SPLINE
SPL {X  -124.054, Y  +777.532, Z    +0.000, E1   -54.436, E3 +80490.887}
SPL {X  -145.922, Y  +742.101, Z    +0.000, E1   -46.535, E3 +80509.157}
SPL {X  -155.216, Y  +715.293, Z    +0.000, E1   -34.460, E3 +80515.349}
SPL {X  -159.282, Y  +691.530, Z    +0.000, E1   -17.100, E3 +80518.044}
SPL {X  -159.981, Y  +678.202, Z    +0.000, E1    -4.129, E3 +80518.618}
SPL {X  -159.990, Y  +674.500, Z    +0.000, E1    +0.000, E3 +80518.655}
SPL {X  -159.990, Y  +672.677, Z    +0.000, E1    +3.879, E3 +80518.671}
SPL {X  -159.990, Y  +669.117, Z    +0.000, E1   +12.900, E3 +80518.754}
SPL {X  -159.990, Y  +665.253, Z    +0.000, E1   +22.908, E3 +80518.927}
SPL {X  -159.990, Y  +658.335, Z    +0.000, E1   +38.839, E3 +80519.472}
SPL {X  -159.990, Y  +645.786, Z    +0.000, E1   +56.338, E3 +80521.186}
SPL {X  -159.990, Y  +623.264, Z    +0.000, E1   +67.753, E3 +80526.112}
SPL {X  -159.990, Y  +547.268, Z    +0.000, E1   +73.735, E3 +80551.800}
SPL {X  -159.626, Y  +366.721, Z    +0.000, E1   +74.756, E3 +80634.065}
SPL {X  -157.975, Y  +352.185, Z    +0.000, E1   +74.622, E3 +80644.131}
SPL {X  -154.546, Y  +336.120, Z    +0.000, E1   +74.400, E3 +80655.790}
SPL {X  -141.909, Y  +303.617, Z    +0.000, E1   +76.515, E3 +80650.757}
ENDSPLINE

SPLINE
SPL {X  -142.567, Y  +304.895, Z    +0.000, E1   +75.566, E3 +80659.572}
ENDSPLINE

SPLINE
SPL {X  -141.999, Y  +303.790, Z    +0.000, E1   +74.633, E3 +80668.823}
SPL {X  -141.780, Y  +303.371, Z    +0.000, E1   +73.549, E3 +80678.397}
SPL {X  -140.619, Y  +301.190, Z    +0.000, E1   +72.741, E3 +80686.243}
SPL {X  -137.438, Y  +295.601, Z    +0.000, E1   +72.365, E3 +80692.332}
SPL {X  -134.156, Y  +290.328, Z    +0.000, E1   +71.962, E3 +80698.203}
SPL {X  -130.677, Y  +285.194, Z    +0.000, E1   +71.519, E3 +80704.008}
SPL {X  -127.147, Y  +280.390, Z    +0.000, E1   +71.042, E3 +80709.492}
SPL {X  -123.431, Y  +275.709, Z    +0.000, E1   +70.518, E3 +80714.815}
SPL {X  -120.392, Y  +272.131, Z    +0.000, E1   +70.053, E3 +80718.835}
SPL {X   -79.311, Y  +238.552, Z    +0.000, E1   +58.563, E3 +80814.074}
ENDSPLINE

SPLINE
SPL {X  -105.077, Y  +256.854, Z    +0.000, E1   +55.187, E3 +81001.627}
SPL {X  -133.208, Y  +288.886, Z    +0.000, E1   +52.003, E3 +81034.728}
SPL {X  -149.825, Y  +321.381, Z    +0.000, E1   +42.580, E3 +81047.881}
SPL {X  -156.491, Y  +344.222, Z    +0.000, E1   +30.612, E3 +81052.387}
SPL {X  -159.275, Y  +362.387, Z    +0.000, E1   +16.907, E3 +81054.301}
SPL {X  -159.964, Y  +374.630, Z    +0.000, E1    +5.249, E3 +81054.875}
SPL {X  -159.990, Y  +379.735, Z    +0.000, E1    -0.236, E3 +81054.932}
SPL {X  -159.990, Y  +384.648, Z    +0.000, E1   -11.739, E3 +81055.028}
SPL {X  -159.990, Y  +391.065, Z    +0.000, E1   -28.187, E3 +81055.356}
SPL {X  -159.990, Y  +397.286, Z    +0.000, E1   -41.591, E3 +81055.899}
SPL {X  -159.990, Y  +406.369, Z    +0.000, E1   -54.148, E3 +81057.118}
SPL {X  -159.990, Y  +426.617, Z    +0.000, E1   -66.230, E3 +81061.367}
SPL {X  -159.990, Y  +499.521, Z    +0.000, E1   -73.662, E3 +81084.694}
SPL {X  -159.629, Y  +687.249, Z    +0.000, E1   -74.539, E3 +81172.578}
SPL {X  -157.983, Y  +701.765, Z    +0.000, E1   -74.384, E3 +81182.810}
SPL {X  -155.520, Y  +714.054, Z    +0.000, E1   -74.151, E3 +81192.564}
SPL {X  -152.569, Y  +724.660, Z    +0.000, E1   -73.857, E3 +81201.799}
SPL {X  -149.625, Y  +733.149, Z    +0.000, E1   -73.553, E3 +81209.734}
SPL {X  -146.617, Y  +740.532, Z    +0.000, E1   -73.233, E3 +81217.011}
SPL {X  -143.394, Y  +747.457, Z    +0.000, E1   -72.883, E3 +81224.108}
SPL {X  -140.332, Y  +753.336, Z    +0.000, E1   -72.527, E3 +81230.383}
SPL {X  -137.187, Y  +758.820, Z    +0.000, E1   -72.156, E3 +81236.386}
SPL {X  -134.014, Y  +763.891, Z    +0.000, E1   -71.759, E3 +81242.071}
SPL {X  -130.657, Y  +768.834, Z    +0.000, E1   -71.330, E3 +81247.687}
SPL {X  -126.937, Y  +773.885, Z    +0.000, E1   -70.823, E3 +81253.488}
SPL {X  -122.983, Y  +778.833, Z    +0.000, E1   -70.262, E3 +81259.133}
SPL {X  -120.205, Y  +782.082, Z    +0.000, E1   -69.822, E3 +81262.801}
SPL {X   -77.717, Y  +816.346, Z    +0.000, E1   -57.422, E3 +81370.653}
SPL {X   -74.440, Y  +818.117, Z    +0.000, E1   -54.647, E3 +81423.892}
ENDSPLINE

SPLINE
SPL {X  -124.054, Y  +777.532, Z    +0.000, E1   -54.436, E3 +81571.968}
SPL {X  -149.719, Y  +732.901, Z    +0.000, E1   -43.150, E3 +81592.782}
SPL {X  -158.004, Y  +701.630, Z    +0.000, E1   -25.366, E3 +81598.247}
SPL {X  -159.838, Y  +683.473, Z    +0.000, E1    -9.532, E3 +81599.554}
SPL {X  -159.990, Y  +674.579, Z    +0.000, E1    -0.168, E3 +81599.736}
SPL {X  -159.990, Y  +672.677, Z    +0.000, E1    +3.879, E3 +81599.752}
SPL {X  -159.990, Y  +669.117, Z    +0.000, E1   +12.900, E3 +81599.835}
SPL {X  -159.990, Y  +663.639, Z    +0.000, E1   +26.675, E3 +81600.120}
SPL {X  -159.990, Y  +656.057, Z    +0.000, E1   +43.288, E3 +81600.776}
SPL {X  -159.990, Y  +645.786, Z    +0.000, E1   +56.338, E3 +81602.267}
SPL {X  -159.990, Y  +623.264, Z    +0.000, E1   +67.753, E3 +81607.193}
SPL {X  -159.990, Y  +547.268, Z    +0.000, E1   +73.735, E3 +81632.881}
SPL {X  -159.626, Y  +366.721, Z    +0.000, E1   +74.756, E3 +81715.146}
SPL {X  -157.975, Y  +352.185, Z    +0.000, E1   +74.622, E3 +81725.212}
SPL {X  -154.546, Y  +336.120, Z    +0.000, E1   +74.400, E3 +81736.871}
SPL {X  -141.909, Y  +303.617, Z    +0.000, E1   +76.515, E3 +81731.838}
ENDSPLINE

SPLINE
SPL {X  -142.567, Y  +304.895, Z    +0.000, E1   +75.566, E3 +81740.653}
ENDSPLINE

SPLINE
SPL {X  -141.999, Y  +303.790, Z    +0.000, E1   +74.633, E3 +81749.904}
SPL {X  -141.780, Y  +303.371, Z    +0.000, E1   +73.549, E3 +81759.478}
SPL {X  -140.619, Y  +301.190, Z    +0.000, E1   +72.741, E3 +81767.324}
SPL {X  -137.438, Y  +295.601, Z    +0.000, E1   +72.365, E3 +81773.413}
SPL {X  -134.156, Y  +290.328, Z    +0.000, E1   +71.962, E3 +81779.284}
SPL {X  -130.677, Y  +285.194, Z    +0.000, E1   +71.519, E3 +81785.089}
SPL {X  -127.147, Y  +280.390, Z    +0.000, E1   +71.042, E3 +81790.573}
SPL {X  -123.431, Y  +275.709, Z    +0.000, E1   +70.518, E3 +81795.896}
SPL {X  -120.392, Y  +272.131, Z    +0.000, E1   +70.053, E3 +81799.916}
SPL {X   -79.311, Y  +238.552, Z    +0.000, E1   +58.563, E3 +81895.155}
ENDSPLINE

SPLINE
SPL {X  -105.077, Y  +256.854, Z    +0.000, E1   +55.187, E3 +82082.708}
SPL {X  -133.208, Y  +288.886, Z    +0.000, E1   +52.003, E3 +82115.809}
SPL {X  -149.825, Y  +321.381, Z    +0.000, E1   +42.580, E3 +82128.962}
SPL {X  -156.491, Y  +344.222, Z    +0.000, E1   +30.612, E3 +82133.468}
SPL {X  -159.275, Y  +362.387, Z    +0.000, E1   +16.907, E3 +82135.382}
SPL {X  -159.964, Y  +374.630, Z    +0.000, E1    +5.249, E3 +82135.956}
SPL {X  -159.990, Y  +379.735, Z    +0.000, E1    -0.236, E3 +82136.013}
SPL {X  -159.990, Y  +384.648, Z    +0.000, E1   -11.739, E3 +82136.109}
SPL {X  -159.990, Y  +389.576, Z    +0.000, E1   -24.732, E3 +82136.336}
SPL {X  -159.990, Y  +395.361, Z    +0.000, E1   -37.740, E3 +82136.794}
SPL {X  -159.990, Y  +406.369, Z    +0.000, E1   -54.148, E3 +82138.199}
SPL {X  -159.990, Y  +426.617, Z    +0.000, E1   -66.230, E3 +82142.448}
SPL {X  -159.990, Y  +499.521, Z    +0.000, E1   -73.662, E3 +82165.775}
SPL {X  -159.629, Y  +687.249, Z    +0.000, E1   -74.539, E3 +82253.659}
SPL {X  -157.983, Y  +701.765, Z    +0.000, E1   -74.384, E3 +82263.891}
SPL {X  -155.520, Y  +714.054, Z    +0.000, E1   -74.151, E3 +82273.646}
SPL {X  -152.569, Y  +724.660, Z    +0.000, E1   -73.857, E3 +82282.880}
SPL {X  -149.625, Y  +733.149, Z    +0.000, E1   -73.553, E3 +82290.815}
SPL {X  -146.617, Y  +740.532, Z    +0.000, E1   -73.233, E3 +82298.092}
SPL {X  -143.394, Y  +747.457, Z    +0.000, E1   -72.883, E3 +82305.189}
SPL {X  -140.332, Y  +753.336, Z    +0.000, E1   -72.527, E3 +82311.464}
SPL {X  -137.187, Y  +758.820, Z    +0.000, E1   -72.156, E3 +82317.467}
SPL {X  -134.014, Y  +763.891, Z    +0.000, E1   -71.759, E3 +82323.152}
SPL {X  -130.657, Y  +768.834, Z    +0.000, E1   -71.330, E3 +82328.768}
SPL {X  -126.937, Y  +773.885, Z    +0.000, E1   -70.823, E3 +82334.569}
SPL {X  -122.983, Y  +778.833, Z    +0.000, E1   -70.262, E3 +82340.214}
SPL {X  -120.205, Y  +782.082, Z    +0.000, E1   -69.822, E3 +82343.882}
SPL {X   -75.772, Y  +817.409, Z    +0.000, E1   -56.226, E3 +82469.821}
ENDSPLINE

SPLINE
SPL {X  -124.054, Y  +777.532, Z    +0.000, E1   -54.436, E3 +82653.049}
SPL {X  -149.719, Y  +732.901, Z    +0.000, E1   -43.150, E3 +82673.863}
SPL {X  -158.004, Y  +701.630, Z    +0.000, E1   -25.366, E3 +82679.328}
SPL {X  -159.639, Y  +687.095, Z    +0.000, E1   -12.931, E3 +82680.486}
SPL {X  -159.981, Y  +678.202, Z    +0.000, E1    -4.129, E3 +82680.780}
SPL {X  -159.990, Y  +674.500, Z    +0.000, E1    +0.000, E3 +82680.818}
SPL {X  -159.990, Y  +672.677, Z    +0.000, E1    +3.879, E3 +82680.833}
SPL {X  -159.990, Y  +669.117, Z    +0.000, E1   +12.900, E3 +82680.916}
SPL {X  -159.990, Y  +663.639, Z    +0.000, E1   +26.675, E3 +82681.201}
SPL {X  -159.990, Y  +656.057, Z    +0.000, E1   +43.288, E3 +82681.857}
SPL {X  -159.990, Y  +645.786, Z    +0.000, E1   +56.338, E3 +82683.348}
SPL {X  -159.990, Y  +623.264, Z    +0.000, E1   +67.753, E3 +82688.274}
SPL {X  -159.990, Y  +547.268, Z    +0.000, E1   +73.735, E3 +82713.962}
SPL {X  -159.091, Y  +360.560, Z    +0.000, E1   +74.726, E3 +82800.289}
SPL {X  -156.418, Y  +343.879, Z    +0.000, E1   +74.473, E3 +82812.714}
SPL {X  -153.414, Y  +332.103, Z    +0.000, E1   +74.378, E3 +82820.389}
SPL {X  -141.909, Y  +303.617, Z    +0.000, E1   +76.515, E3 +82812.919}
ENDSPLINE

SPLINE
SPL {X  -142.567, Y  +304.895, Z    +0.000, E1   +75.566, E3 +82821.734}
ENDSPLINE

SPLINE
SPL {X  -141.999, Y  +303.790, Z    +0.000, E1   +74.633, E3 +82830.985}
SPL {X  -141.780, Y  +303.371, Z    +0.000, E1   +73.549, E3 +82840.559}
SPL {X  -140.619, Y  +301.190, Z    +0.000, E1   +72.741, E3 +82848.406}
SPL {X  -137.438, Y  +295.601, Z    +0.000, E1   +72.365, E3 +82854.494}
SPL {X  -134.156, Y  +290.328, Z    +0.000, E1   +71.962, E3 +82860.365}
SPL {X  -130.677, Y  +285.194, Z    +0.000, E1   +71.519, E3 +82866.170}
SPL {X  -126.239, Y  +279.212, Z    +0.000, E1   +70.937, E3 +82872.971}
SPL {X  -121.335, Y  +273.218, Z    +0.000, E1   +70.225, E3 +82879.759}
SPL {X   -79.311, Y  +238.552, Z    +0.000, E1   +58.563, E3 +82976.236}
ENDSPLINE

SPLINE
SPL {X  -105.077, Y  +256.854, Z    +0.000, E1   +55.187, E3 +83163.789}
SPL {X  -133.208, Y  +288.886, Z    +0.000, E1   +52.003, E3 +83196.890}
SPL {X  -149.825, Y  +321.381, Z    +0.000, E1   +42.580, E3 +83210.043}
SPL {X  -156.491, Y  +344.222, Z    +0.000, E1   +30.612, E3 +83214.549}
SPL {X  -159.275, Y  +362.387, Z    +0.000, E1   +16.907, E3 +83216.463}
SPL {X  -159.964, Y  +374.630, Z    +0.000, E1    +5.249, E3 +83217.037}
SPL {X  -159.990, Y  +379.484, Z    +0.000, E1    +0.034, E3 +83217.093}
SPL {X  -159.990, Y  +381.639, Z    +0.000, E1    -4.454, E3 +83217.114}
SPL {X  -159.990, Y  +385.871, Z    +0.000, E1   -15.161, E3 +83217.230}
SPL {X  -159.990, Y  +391.065, Z    +0.000, E1   -28.187, E3 +83217.518}
SPL {X  -159.990, Y  +397.286, Z    +0.000, E1   -41.591, E3 +83218.061}
SPL {X  -159.990, Y  +406.369, Z    +0.000, E1   -54.148, E3 +83219.280}
SPL {X  -159.990, Y  +426.617, Z    +0.000, E1   -66.230, E3 +83223.530}
SPL {X  -159.990, Y  +499.521, Z    +0.000, E1   -73.662, E3 +83246.856}
SPL {X  -159.629, Y  +687.249, Z    +0.000, E1   -74.539, E3 +83334.740}
SPL {X  -157.983, Y  +701.765, Z    +0.000, E1   -74.384, E3 +83344.973}
SPL {X  -155.520, Y  +714.054, Z    +0.000, E1   -74.151, E3 +83354.727}
SPL {X  -152.569, Y  +724.660, Z    +0.000, E1   -73.857, E3 +83363.961}
SPL {X  -149.625, Y  +733.149, Z    +0.000, E1   -73.553, E3 +83371.896}
SPL {X  -146.617, Y  +740.532, Z    +0.000, E1   -73.233, E3 +83379.173}
SPL {X  -143.394, Y  +747.457, Z    +0.000, E1   -72.883, E3 +83386.270}
SPL {X  -140.332, Y  +753.336, Z    +0.000, E1   -72.527, E3 +83392.545}
SPL {X  -137.187, Y  +758.820, Z    +0.000, E1   -72.156, E3 +83398.548}
SPL {X  -134.014, Y  +763.891, Z    +0.000, E1   -71.759, E3 +83404.233}
SPL {X  -130.657, Y  +768.834, Z    +0.000, E1   -71.330, E3 +83409.849}
SPL {X  -126.020, Y  +775.068, Z    +0.000, E1   -70.718, E3 +83416.976}
SPL {X  -121.287, Y  +780.838, Z    +0.000, E1   -70.013, E3 +83423.550}
SPL {X   -75.772, Y  +817.409, Z    +0.000, E1   -56.226, E3 +83550.902}
ENDSPLINE

SPLINE
SPL {X  -124.054, Y  +777.532, Z    +0.000, E1   -54.436, E3 +83734.130}
SPL {X  -149.719, Y  +732.901, Z    +0.000, E1   -43.150, E3 +83754.944}
SPL {X  -158.004, Y  +701.630, Z    +0.000, E1   -25.366, E3 +83760.409}
SPL {X  -159.639, Y  +687.095, Z    +0.000, E1   -12.931, E3 +83761.567}
SPL {X  -159.981, Y  +678.202, Z    +0.000, E1    -4.129, E3 +83761.861}
SPL {X  -159.990, Y  +674.500, Z    +0.000, E1    +0.000, E3 +83761.899}
SPL {X  -159.990, Y  +672.677, Z    +0.000, E1    +3.879, E3 +83761.914}
SPL {X  -159.990, Y  +669.117, Z    +0.000, E1   +12.900, E3 +83761.997}
SPL {X  -159.990, Y  +663.639, Z    +0.000, E1   +26.675, E3 +83762.282}
SPL {X  -159.990, Y  +656.057, Z    +0.000, E1   +43.288, E3 +83762.938}
SPL {X  -159.990, Y  +645.786, Z    +0.000, E1   +56.338, E3 +83764.429}
SPL {X  -159.990, Y  +623.264, Z    +0.000, E1   +67.753, E3 +83769.355}
SPL {X  -159.990, Y  +547.268, Z    +0.000, E1   +73.735, E3 +83795.043}
SPL {X  -159.091, Y  +360.560, Z    +0.000, E1   +74.726, E3 +83881.370}
SPL {X  -156.418, Y  +343.879, Z    +0.000, E1   +74.473, E3 +83893.795}
SPL {X  -153.414, Y  +332.103, Z    +0.000, E1   +74.378, E3 +83901.470}
SPL {X  -141.909, Y  +303.617, Z    +0.000, E1   +76.515, E3 +83894.000}
ENDSPLINE

SPLINE
SPL {X  -142.567, Y  +304.895, Z    +0.000, E1   +75.566, E3 +83902.815}
ENDSPLINE

SPLINE
SPL {X  -141.999, Y  +303.790, Z    +0.000, E1   +74.633, E3 +83912.066}
SPL {X  -141.780, Y  +303.371, Z    +0.000, E1   +73.549, E3 +83921.640}
SPL {X  -140.619, Y  +301.190, Z    +0.000, E1   +72.741, E3 +83929.487}
SPL {X  -137.438, Y  +295.601, Z    +0.000, E1   +72.365, E3 +83935.575}
SPL {X  -134.156, Y  +290.328, Z    +0.000, E1   +71.962, E3 +83941.446}
SPL {X  -130.677, Y  +285.194, Z    +0.000, E1   +71.519, E3 +83947.251}
SPL {X  -127.147, Y  +280.390, Z    +0.000, E1   +71.042, E3 +83952.735}
SPL {X  -123.431, Y  +275.709, Z    +0.000, E1   +70.518, E3 +83958.058}
SPL {X  -120.392, Y  +272.131, Z    +0.000, E1   +70.053, E3 +83962.078}
SPL {X   -79.311, Y  +238.552, Z    +0.000, E1   +58.563, E3 +84057.317}
ENDSPLINE

SPLINE
SPL {X  -105.077, Y  +256.854, Z    +0.000, E1   +55.187, E3 +84244.870}
SPL {X  -133.208, Y  +288.886, Z    +0.000, E1   +52.003, E3 +84277.971}
SPL {X  -149.825, Y  +321.381, Z    +0.000, E1   +42.580, E3 +84291.124}
SPL {X  -157.376, Y  +348.695, Z    +0.000, E1   +27.651, E3 +84296.209}
SPL {X  -159.486, Y  +364.808, Z    +0.000, E1   +14.693, E3 +84297.713}
SPL {X  -159.964, Y  +374.630, Z    +0.000, E1    +5.249, E3 +84298.118}
SPL {X  -159.990, Y  +379.484, Z    +0.000, E1    +0.034, E3 +84298.174}
SPL {X  -159.990, Y  +381.639, Z    +0.000, E1    -4.454, E3 +84298.195}
SPL {X  -159.990, Y  +385.871, Z    +0.000, E1   -15.161, E3 +84298.311}
SPL {X  -159.990, Y  +391.065, Z    +0.000, E1   -28.187, E3 +84298.599}
SPL {X  -159.990, Y  +399.326, Z    +0.000, E1   -44.934, E3 +84299.383}
SPL {X  -159.990, Y  +408.817, Z    +0.000, E1   -56.572, E3 +84300.755}
SPL {X  -159.990, Y  +426.617, Z    +0.000, E1   -66.230, E3 +84304.611}
SPL {X  -159.990, Y  +499.521, Z    +0.000, E1   -73.662, E3 +84327.937}
SPL {X  -159.629, Y  +687.249, Z    +0.000, E1   -74.539, E3 +84415.821}
SPL {X  -157.983, Y  +701.765, Z    +0.000, E1   -74.384, E3 +84426.054}
SPL {X  -155.520, Y  +714.054, Z    +0.000, E1   -74.151, E3 +84435.808}
SPL {X  -152.569, Y  +724.660, Z    +0.000, E1   -73.857, E3 +84445.042}
SPL {X  -149.625, Y  +733.149, Z    +0.000, E1   -73.553, E3 +84452.977}
SPL {X  -146.617, Y  +740.532, Z    +0.000, E1   -73.233, E3 +84460.254}
SPL {X  -143.394, Y  +747.457, Z    +0.000, E1   -72.883, E3 +84467.351}
SPL {X  -140.332, Y  +753.336, Z    +0.000, E1   -72.527, E3 +84473.626}
SPL {X  -137.187, Y  +758.820, Z    +0.000, E1   -72.156, E3 +84479.629}
SPL {X  -134.014, Y  +763.891, Z    +0.000, E1   -71.759, E3 +84485.314}
SPL {X  -129.643, Y  +770.252, Z    +0.000, E1   -71.218, E3 +84492.521}
SPL {X  -125.230, Y  +776.071, Z    +0.000, E1   -70.580, E3 +84499.240}
SPL {X  -122.263, Y  +779.692, Z    +0.000, E1   -70.136, E3 +84503.369}
SPL {X  -120.205, Y  +782.082, Z    +0.000, E1   -69.822, E3 +84506.044}
SPL {X   -75.772, Y  +817.409, Z    +0.000, E1   -56.226, E3 +84631.983}
ENDSPLINE

SPLINE
SPL {X  -124.054, Y  +777.532, Z    +0.000, E1   -54.436, E3 +84815.211}
SPL {X  -145.922, Y  +742.101, Z    +0.000, E1   -46.535, E3 +84833.481}
SPL {X  -155.216, Y  +715.293, Z    +0.000, E1   -34.460, E3 +84839.673}
SPL {X  -158.715, Y  +696.660, Z    +0.000, E1   -21.368, E3 +84842.001}
SPL {X  -159.639, Y  +687.095, Z    +0.000, E1   -12.931, E3 +84842.648}
SPL {X  -159.981, Y  +678.202, Z    +0.000, E1    -4.129, E3 +84842.942}
SPL {X  -159.990, Y  +674.500, Z    +0.000, E1    +0.000, E3 +84842.980}
SPL {X  -159.990, Y  +672.677, Z    +0.000, E1    +3.879, E3 +84842.995}
SPL {X  -159.990, Y  +669.117, Z    +0.000, E1   +12.900, E3 +84843.078}
SPL {X  -159.990, Y  +663.639, Z    +0.000, E1   +26.675, E3 +84843.363}
SPL {X  -159.990, Y  +656.057, Z    +0.000, E1   +43.288, E3 +84844.019}
SPL {X  -159.990, Y  +647.797, Z    +0.000, E1   +54.469, E3 +84845.156}
SPL {X  -159.990, Y  +630.178, Z    +0.000, E1   +65.480, E3 +84848.840}
SPL {X  -159.990, Y  +547.268, Z    +0.000, E1   +73.735, E3 +84876.124}
SPL {X  -159.626, Y  +366.721, Z    +0.000, E1   +74.756, E3 +84958.390}
SPL {X  -158.582, Y  +356.317, Z    +0.000, E1   +74.662, E3 +84965.483}
SPL {X  -156.418, Y  +343.879, Z    +0.000, E1   +74.473, E3 +84974.876}
SPL {X  -153.414, Y  +332.103, Z    +0.000, E1   +74.378, E3 +84982.551}
SPL {X  -141.909, Y  +303.617, Z    +0.000, E1   +76.515, E3 +84975.081}
ENDSPLINE

SPLINE
SPL {X  -142.567, Y  +304.895, Z    +0.000, E1   +75.566, E3 +84983.896}
ENDSPLINE

SPLINE
SPL {X  -141.999, Y  +303.790, Z    +0.000, E1   +74.633, E3 +84993.147}
SPL {X  -141.780, Y  +303.371, Z    +0.000, E1   +73.549, E3 +85002.721}
SPL {X  -140.619, Y  +301.190, Z    +0.000, E1   +72.741, E3 +85010.568}
SPL {X  -137.438, Y  +295.601, Z    +0.000, E1   +72.365, E3 +85016.656}
SPL {X  -134.156, Y  +290.328, Z    +0.000, E1   +71.962, E3 +85022.527}
SPL {X  -130.677, Y  +285.194, Z    +0.000, E1   +71.519, E3 +85028.332}
SPL {X  -127.147, Y  +280.390, Z    +0.000, E1   +71.042, E3 +85033.816}
SPL {X  -123.431, Y  +275.709, Z    +0.000, E1   +70.518, E3 +85039.139}
SPL {X  -120.392, Y  +272.131, Z    +0.000, E1   +70.053, E3 +85043.160}
SPL {X   -79.311, Y  +238.552, Z    +0.000, E1   +58.563, E3 +85138.399}
ENDSPLINE

SPLINE
SPL {X  -105.077, Y  +256.854, Z    +0.000, E1   +55.187, E3 +85325.951}
SPL {X  -133.208, Y  +288.886, Z    +0.000, E1   +52.003, E3 +85359.052}
SPL {X  -149.825, Y  +321.381, Z    +0.000, E1   +42.580, E3 +85372.205}
SPL {X  -157.376, Y  +348.695, Z    +0.000, E1   +27.651, E3 +85377.290}
SPL {X  -159.486, Y  +364.808, Z    +0.000, E1   +14.693, E3 +85378.794}
SPL {X  -159.964, Y  +374.630, Z    +0.000, E1    +5.249, E3 +85379.199}
SPL {X  -159.990, Y  +379.484, Z    +0.000, E1    +0.034, E3 +85379.255}
SPL {X  -159.990, Y  +381.639, Z    +0.000, E1    -4.454, E3 +85379.276}
SPL {X  -159.990, Y  +385.871, Z    +0.000, E1   -15.161, E3 +85379.392}
SPL {X  -159.990, Y  +391.065, Z    +0.000, E1   -28.187, E3 +85379.680}
SPL {X  -159.990, Y  +399.326, Z    +0.000, E1   -44.934, E3 +85380.464}
SPL {X  -159.990, Y  +408.817, Z    +0.000, E1   -56.572, E3 +85381.836}
SPL {X  -159.990, Y  +426.617, Z    +0.000, E1   -66.230, E3 +85385.692}
SPL {X  -159.990, Y  +499.521, Z    +0.000, E1   -73.662, E3 +85409.018}
SPL {X  -159.629, Y  +687.249, Z    +0.000, E1   -74.539, E3 +85496.902}
SPL {X  -157.983, Y  +701.765, Z    +0.000, E1   -74.384, E3 +85507.135}
SPL {X  -155.520, Y  +714.054, Z    +0.000, E1   -74.151, E3 +85516.889}
SPL {X  -152.569, Y  +724.660, Z    +0.000, E1   -73.857, E3 +85526.123}
SPL {X  -149.625, Y  +733.149, Z    +0.000, E1   -73.553, E3 +85534.059}
SPL {X  -146.617, Y  +740.532, Z    +0.000, E1   -73.233, E3 +85541.335}
SPL {X  -143.394, Y  +747.457, Z    +0.000, E1   -72.883, E3 +85548.432}
SPL {X  -140.332, Y  +753.336, Z    +0.000, E1   -72.527, E3 +85554.707}
SPL {X  -137.187, Y  +758.820, Z    +0.000, E1   -72.156, E3 +85560.710}
SPL {X  -134.014, Y  +763.891, Z    +0.000, E1   -71.759, E3 +85566.396}
SPL {X  -129.643, Y  +770.252, Z    +0.000, E1   -71.218, E3 +85573.602}
SPL {X  -125.230, Y  +776.071, Z    +0.000, E1   -70.580, E3 +85580.321}
SPL {X  -121.287, Y  +780.838, Z    +0.000, E1   -70.013, E3 +85585.712}
SPL {X   -75.772, Y  +817.409, Z    +0.000, E1   -56.226, E3 +85713.064}
ENDSPLINE

SPLINE
SPL {X  -124.054, Y  +777.532, Z    +0.000, E1   -54.436, E3 +85896.292}
SPL {X  -145.922, Y  +742.101, Z    +0.000, E1   -46.535, E3 +85914.562}
SPL {X  -155.216, Y  +715.293, Z    +0.000, E1   -34.460, E3 +85920.754}
SPL {X  -158.715, Y  +696.660, Z    +0.000, E1   -21.368, E3 +85923.082}
SPL {X  -159.838, Y  +683.473, Z    +0.000, E1    -9.532, E3 +85923.878}
SPL {X  -159.990, Y  +674.579, Z    +0.000, E1    -0.168, E3 +85924.061}
SPL {X  -159.990, Y  +672.677, Z    +0.000, E1    +3.879, E3 +85924.076}
SPL {X  -159.990, Y  +669.117, Z    +0.000, E1   +12.900, E3 +85924.159}
SPL {X  -159.990, Y  +663.639, Z    +0.000, E1   +26.675, E3 +85924.445}
SPL {X  -159.990, Y  +656.057, Z    +0.000, E1   +43.288, E3 +85925.100}
SPL {X  -159.990, Y  +647.797, Z    +0.000, E1   +54.469, E3 +85926.238}
SPL {X  -159.990, Y  +630.178, Z    +0.000, E1   +65.480, E3 +85929.921}
SPL {X  -159.990, Y  +547.268, Z    +0.000, E1   +73.735, E3 +85957.206}
SPL {X  -159.091, Y  +360.560, Z    +0.000, E1   +74.726, E3 +86043.532}
SPL {X  -156.418, Y  +343.879, Z    +0.000, E1   +74.473, E3 +86055.957}
SPL {X  -153.414, Y  +332.103, Z    +0.000, E1   +74.378, E3 +86063.632}
SPL {X  -141.909, Y  +303.617, Z    +0.000, E1   +76.515, E3 +86056.162}
ENDSPLINE

SPLINE
SPL {X  -142.567, Y  +304.895, Z    +0.000, E1   +75.566, E3 +86064.977}
ENDSPLINE

SPLINE
SPL {X  -141.999, Y  +303.790, Z    +0.000, E1   +74.633, E3 +86074.228}
SPL {X  -141.780, Y  +303.371, Z    +0.000, E1   +73.549, E3 +86083.802}
SPL {X  -140.619, Y  +301.190, Z    +0.000, E1   +72.741, E3 +86091.649}
SPL {X  -137.438, Y  +295.601, Z    +0.000, E1   +72.365, E3 +86097.737}
SPL {X  -134.156, Y  +290.328, Z    +0.000, E1   +71.962, E3 +86103.608}
SPL {X  -130.677, Y  +285.194, Z    +0.000, E1   +71.519, E3 +86109.413}
SPL {X  -127.147, Y  +280.390, Z    +0.000, E1   +71.042, E3 +86114.897}
SPL {X  -123.431, Y  +275.709, Z    +0.000, E1   +70.518, E3 +86120.220}
SPL {X  -120.392, Y  +272.131, Z    +0.000, E1   +70.053, E3 +86124.241}
SPL {X   -79.311, Y  +238.552, Z    +0.000, E1   +58.563, E3 +86219.480}
ENDSPLINE

SPLINE
SPL {X  -105.077, Y  +256.854, Z    +0.000, E1   +55.187, E3 +86407.032}
SPL {X  -133.208, Y  +288.886, Z    +0.000, E1   +52.003, E3 +86440.133}
SPL {X  -149.825, Y  +321.381, Z    +0.000, E1   +42.580, E3 +86453.287}
SPL {X  -156.491, Y  +344.222, Z    +0.000, E1   +30.612, E3 +86457.793}
SPL {X  -159.275, Y  +362.387, Z    +0.000, E1   +16.907, E3 +86459.707}
SPL {X  -159.964, Y  +374.630, Z    +0.000, E1    +5.249, E3 +86460.280}
SPL {X  -159.990, Y  +379.735, Z    +0.000, E1    -0.236, E3 +86460.337}
SPL {X  -159.990, Y  +384.648, Z    +0.000, E1   -11.739, E3 +86460.434}
SPL {X  -159.990, Y  +391.065, Z    +0.000, E1   -28.187, E3 +86460.761}
SPL {X  -159.990, Y  +397.286, Z    +0.000, E1   -41.591, E3 +86461.304}
SPL {X  -159.990, Y  +406.369, Z    +0.000, E1   -54.148, E3 +86462.523}
SPL {X  -159.990, Y  +426.617, Z    +0.000, E1   -66.230, E3 +86466.773}
SPL {X  -159.990, Y  +499.521, Z    +0.000, E1   -73.662, E3 +86490.099}
SPL {X  -159.629, Y  +687.249, Z    +0.000, E1   -74.539, E3 +86577.984}
SPL {X  -157.983, Y  +701.765, Z    +0.000, E1   -74.384, E3 +86588.216}
SPL {X  -155.520, Y  +714.054, Z    +0.000, E1   -74.151, E3 +86597.970}
SPL {X  -152.569, Y  +724.660, Z    +0.000, E1   -73.857, E3 +86607.204}
SPL {X  -149.625, Y  +733.149, Z    +0.000, E1   -73.553, E3 +86615.140}
SPL {X  -146.617, Y  +740.532, Z    +0.000, E1   -73.233, E3 +86622.416}
SPL {X  -143.394, Y  +747.457, Z    +0.000, E1   -72.883, E3 +86629.513}
SPL {X  -140.332, Y  +753.336, Z    +0.000, E1   -72.527, E3 +86635.788}
SPL {X  -137.187, Y  +758.820, Z    +0.000, E1   -72.156, E3 +86641.791}
SPL {X  -134.014, Y  +763.891, Z    +0.000, E1   -71.759, E3 +86647.477}
SPL {X  -129.643, Y  +770.252, Z    +0.000, E1   -71.218, E3 +86654.683}
SPL {X  -125.230, Y  +776.071, Z    +0.000, E1   -70.580, E3 +86661.402}
SPL {X  -122.263, Y  +779.692, Z    +0.000, E1   -70.136, E3 +86665.531}
SPL {X  -120.205, Y  +782.082, Z    +0.000, E1   -69.822, E3 +86668.207}
SPL {X   -77.717, Y  +816.346, Z    +0.000, E1   -57.422, E3 +86776.058}
SPL {X   -74.440, Y  +818.117, Z    +0.000, E1   -54.647, E3 +86829.297}
ENDSPLINE

SPLINE
SPL {X  -124.054, Y  +777.532, Z    +0.000, E1   -54.436, E3 +86977.373}
SPL {X  -149.719, Y  +732.901, Z    +0.000, E1   -43.150, E3 +86998.188}
SPL {X  -158.004, Y  +701.630, Z    +0.000, E1   -25.366, E3 +87003.652}
SPL {X  -159.639, Y  +687.095, Z    +0.000, E1   -12.931, E3 +87004.811}
SPL {X  -159.981, Y  +678.202, Z    +0.000, E1    -4.129, E3 +87005.104}
SPL {X  -159.990, Y  +674.500, Z    +0.000, E1    +0.000, E3 +87005.142}
SPL {X  -159.990, Y  +672.677, Z    +0.000, E1    +3.879, E3 +87005.157}
SPL {X  -159.990, Y  +669.117, Z    +0.000, E1   +12.900, E3 +87005.240}
SPL {X  -159.990, Y  +663.639, Z    +0.000, E1   +26.675, E3 +87005.526}
SPL {X  -159.990, Y  +656.057, Z    +0.000, E1   +43.288, E3 +87006.181}
SPL {X  -159.990, Y  +647.797, Z    +0.000, E1   +54.469, E3 +87007.319}
SPL {X  -159.990, Y  +630.178, Z    +0.000, E1   +65.480, E3 +87011.002}
SPL {X  -159.990, Y  +547.268, Z    +0.000, E1   +73.735, E3 +87038.287}
SPL {X  -159.626, Y  +366.721, Z    +0.000, E1   +74.756, E3 +87120.552}
SPL {X  -158.582, Y  +356.317, Z    +0.000, E1   +74.662, E3 +87127.645}
SPL {X  -156.418, Y  +343.879, Z    +0.000, E1   +74.473, E3 +87137.038}
SPL {X  -153.414, Y  +332.103, Z    +0.000, E1   +74.378, E3 +87144.713}
SPL {X  -141.909, Y  +303.617, Z    +0.000, E1   +76.515, E3 +87137.243}
ENDSPLINE

SPLINE
SPL {X  -142.567, Y  +304.895, Z    +0.000, E1   +75.566, E3 +87146.058}
ENDSPLINE

SPLINE
SPL {X  -141.999, Y  +303.790, Z    +0.000, E1   +74.633, E3 +87155.309}
SPL {X  -141.780, Y  +303.371, Z    +0.000, E1   +73.549, E3 +87164.883}
SPL {X  -140.619, Y  +301.190, Z    +0.000, E1   +72.741, E3 +87172.730}
SPL {X  -137.438, Y  +295.601, Z    +0.000, E1   +72.365, E3 +87178.818}
SPL {X  -134.156, Y  +290.328, Z    +0.000, E1   +71.962, E3 +87184.689}
SPL {X  -130.677, Y  +285.194, Z    +0.000, E1   +71.519, E3 +87190.494}
SPL {X  -127.147, Y  +280.390, Z    +0.000, E1   +71.042, E3 +87195.978}
SPL {X  -123.431, Y  +275.709, Z    +0.000, E1   +70.518, E3 +87201.301}
SPL {X  -120.392, Y  +272.131, Z    +0.000, E1   +70.053, E3 +87205.322}
SPL {X   -79.311, Y  +238.552, Z    +0.000, E1   +58.563, E3 +87300.561}
ENDSPLINE

SPLINE
SPL {X  -105.077, Y  +256.854, Z    +0.000, E1   +55.187, E3 +87488.113}
SPL {X  -133.208, Y  +288.886, Z    +0.000, E1   +52.003, E3 +87521.214}
SPL {X  -149.825, Y  +321.381, Z    +0.000, E1   +42.580, E3 +87534.368}
SPL {X  -157.376, Y  +348.695, Z    +0.000, E1   +27.651, E3 +87539.453}
SPL {X  -159.486, Y  +364.808, Z    +0.000, E1   +14.693, E3 +87540.956}
SPL {X  -159.964, Y  +374.630, Z    +0.000, E1    +5.249, E3 +87541.361}
SPL {X  -159.990, Y  +379.735, Z    +0.000, E1    -0.236, E3 +87541.418}
SPL {X  -159.990, Y  +384.648, Z    +0.000, E1   -11.739, E3 +87541.515}
SPL {X  -159.990, Y  +391.065, Z    +0.000, E1   -28.187, E3 +87541.843}
SPL {X  -159.990, Y  +397.286, Z    +0.000, E1   -41.591, E3 +87542.385}
SPL {X  -159.990, Y  +406.369, Z    +0.000, E1   -54.148, E3 +87543.604}
SPL {X  -159.990, Y  +426.617, Z    +0.000, E1   -66.230, E3 +87547.854}
SPL {X  -159.990, Y  +499.521, Z    +0.000, E1   -73.662, E3 +87571.180}
SPL {X  -159.629, Y  +687.249, Z    +0.000, E1   -74.539, E3 +87659.065}
SPL {X  -157.983, Y  +701.765, Z    +0.000, E1   -74.384, E3 +87669.297}
SPL {X  -155.520, Y  +714.054, Z    +0.000, E1   -74.151, E3 +87679.051}
SPL {X  -152.569, Y  +724.660, Z    +0.000, E1   -73.857, E3 +87688.286}
SPL {X  -149.625, Y  +733.149, Z    +0.000, E1   -73.553, E3 +87696.221}
SPL {X  -146.617, Y  +740.532, Z    +0.000, E1   -73.233, E3 +87703.497}
SPL {X  -143.394, Y  +747.457, Z    +0.000, E1   -72.883, E3 +87710.594}
SPL {X  -140.332, Y  +753.336, Z    +0.000, E1   -72.527, E3 +87716.869}
SPL {X  -137.187, Y  +758.820, Z    +0.000, E1   -72.156, E3 +87722.872}
SPL {X  -134.014, Y  +763.891, Z    +0.000, E1   -71.759, E3 +87728.558}
SPL {X  -130.657, Y  +768.834, Z    +0.000, E1   -71.330, E3 +87734.173}
SPL {X  -126.020, Y  +775.068, Z    +0.000, E1   -70.718, E3 +87741.301}
SPL {X  -121.287, Y  +780.838, Z    +0.000, E1   -70.013, E3 +87747.874}
SPL {X   -75.772, Y  +817.409, Z    +0.000, E1   -56.226, E3 +87875.227}
ENDSPLINE

SPLINE
SPL {X  -124.054, Y  +777.532, Z    +0.000, E1   -54.436, E3 +88058.454}
SPL {X  -149.719, Y  +732.901, Z    +0.000, E1   -43.150, E3 +88079.269}
SPL {X  -158.004, Y  +701.630, Z    +0.000, E1   -25.366, E3 +88084.733}
SPL {X  -159.639, Y  +687.095, Z    +0.000, E1   -12.931, E3 +88085.892}
SPL {X  -159.981, Y  +678.202, Z    +0.000, E1    -4.129, E3 +88086.185}
SPL {X  -159.990, Y  +674.500, Z    +0.000, E1    +0.000, E3 +88086.223}
SPL {X  -159.990, Y  +672.677, Z    +0.000, E1    +3.879, E3 +88086.238}
SPL {X  -159.990, Y  +669.117, Z    +0.000, E1   +12.900, E3 +88086.321}
SPL {X  -159.990, Y  +663.639, Z    +0.000, E1   +26.675, E3 +88086.607}
SPL {X  -159.990, Y  +656.057, Z    +0.000, E1   +43.288, E3 +88087.262}
SPL {X  -159.990, Y  +645.786, Z    +0.000, E1   +56.338, E3 +88088.754}
SPL {X  -159.990, Y  +623.264, Z    +0.000, E1   +67.753, E3 +88093.680}
SPL {X  -159.990, Y  +547.268, Z    +0.000, E1   +73.735, E3 +88119.368}
SPL {X  -159.091, Y  +360.560, Z    +0.000, E1   +74.726, E3 +88205.694}
SPL {X  -156.418, Y  +343.879, Z    +0.000, E1   +74.473, E3 +88218.119}
SPL {X  -153.414, Y  +332.103, Z    +0.000, E1   +74.378, E3 +88225.794}
SPL {X  -141.909, Y  +303.617, Z    +0.000, E1   +76.515, E3 +88218.324}
ENDSPLINE

SPLINE
SPL {X  -142.567, Y  +304.895, Z    +0.000, E1   +75.566, E3 +88227.139}
ENDSPLINE

SPLINE
SPL {X  -141.999, Y  +303.790, Z    +0.000, E1   +74.633, E3 +88236.391}
SPL {X  -141.780, Y  +303.371, Z    +0.000, E1   +73.549, E3 +88245.964}
SPL {X  -140.619, Y  +301.190, Z    +0.000, E1   +72.741, E3 +88253.811}
SPL {X  -137.438, Y  +295.601, Z    +0.000, E1   +72.365, E3 +88259.899}
SPL {X  -134.156, Y  +290.328, Z    +0.000, E1   +71.962, E3 +88265.770}
SPL {X  -130.677, Y  +285.194, Z    +0.000, E1   +71.519, E3 +88271.575}
SPL {X  -126.239, Y  +279.212, Z    +0.000, E1   +70.937, E3 +88278.376}
SPL {X  -121.335, Y  +273.218, Z    +0.000, E1   +70.225, E3 +88285.164}
SPL {X   -79.311, Y  +238.552, Z    +0.000, E1   +58.563, E3 +88381.642}
ENDSPLINE

SPLINE
SPL {X  -105.077, Y  +256.854, Z    +0.000, E1   +55.187, E3 +88569.194}
SPL {X  -133.208, Y  +288.886, Z    +0.000, E1   +52.003, E3 +88602.295}
SPL {X  -149.825, Y  +321.381, Z    +0.000, E1   +42.580, E3 +88615.449}
SPL {X  -156.491, Y  +344.222, Z    +0.000, E1   +30.612, E3 +88619.955}
SPL {X  -159.275, Y  +362.387, Z    +0.000, E1   +16.907, E3 +88621.869}
SPL {X  -159.964, Y  +374.630, Z    +0.000, E1    +5.249, E3 +88622.442}
SPL {X  -159.990, Y  +379.484, Z    +0.000, E1    +0.034, E3 +88622.498}
SPL {X  -159.990, Y  +381.639, Z    +0.000, E1    -4.454, E3 +88622.520}
SPL {X  -159.990, Y  +385.871, Z    +0.000, E1   -15.161, E3 +88622.636}
SPL {X  -159.990, Y  +391.065, Z    +0.000, E1   -28.187, E3 +88622.924}
SPL {X  -159.990, Y  +397.286, Z    +0.000, E1   -41.591, E3 +88623.466}
SPL {X  -159.990, Y  +406.369, Z    +0.000, E1   -54.148, E3 +88624.685}
SPL {X  -159.990, Y  +426.617, Z    +0.000, E1   -66.230, E3 +88628.935}
SPL {X  -159.990, Y  +499.521, Z    +0.000, E1   -73.662, E3 +88652.262}
SPL {X  -159.629, Y  +687.249, Z    +0.000, E1   -74.539, E3 +88740.146}
SPL {X  -157.983, Y  +701.765, Z    +0.000, E1   -74.384, E3 +88750.378}
SPL {X  -155.520, Y  +714.054, Z    +0.000, E1   -74.151, E3 +88760.132}
SPL {X  -152.569, Y  +724.660, Z    +0.000, E1   -73.857, E3 +88769.367}
SPL {X  -149.625, Y  +733.149, Z    +0.000, E1   -73.553, E3 +88777.302}
SPL {X  -146.617, Y  +740.532, Z    +0.000, E1   -73.233, E3 +88784.578}
SPL {X  -143.394, Y  +747.457, Z    +0.000, E1   -72.883, E3 +88791.675}
SPL {X  -140.332, Y  +753.336, Z    +0.000, E1   -72.527, E3 +88797.950}
SPL {X  -137.187, Y  +758.820, Z    +0.000, E1   -72.156, E3 +88803.953}
SPL {X  -134.014, Y  +763.891, Z    +0.000, E1   -71.759, E3 +88809.639}
SPL {X  -130.657, Y  +768.834, Z    +0.000, E1   -71.330, E3 +88815.254}
SPL {X  -126.937, Y  +773.885, Z    +0.000, E1   -70.823, E3 +88821.056}
SPL {X  -122.983, Y  +778.833, Z    +0.000, E1   -70.262, E3 +88826.701}
SPL {X  -120.205, Y  +782.082, Z    +0.000, E1   -69.822, E3 +88830.369}
SPL {X   -75.772, Y  +817.409, Z    +0.000, E1   -56.226, E3 +88956.308}
ENDSPLINE

SPLINE
SPL {X  -124.054, Y  +777.532, Z    +0.000, E1   -54.436, E3 +89139.535}
SPL {X  -145.922, Y  +742.101, Z    +0.000, E1   -46.535, E3 +89157.805}
SPL {X  -155.216, Y  +715.293, Z    +0.000, E1   -34.460, E3 +89163.998}
SPL {X  -159.282, Y  +691.530, Z    +0.000, E1   -17.100, E3 +89166.693}
SPL {X  -159.981, Y  +678.202, Z    +0.000, E1    -4.129, E3 +89167.267}
SPL {X  -159.990, Y  +674.500, Z    +0.000, E1    +0.000, E3 +89167.304}
SPL {X  -159.990, Y  +672.677, Z    +0.000, E1    +3.879, E3 +89167.319}
SPL {X  -159.990, Y  +669.117, Z    +0.000, E1   +12.900, E3 +89167.402}
SPL {X  -159.990, Y  +665.253, Z    +0.000, E1   +22.908, E3 +89167.576}
SPL {X  -159.990, Y  +658.335, Z    +0.000, E1   +38.839, E3 +89168.121}
SPL {X  -159.990, Y  +645.786, Z    +0.000, E1   +56.338, E3 +89169.835}
SPL {X  -159.990, Y  +623.264, Z    +0.000, E1   +67.753, E3 +89174.761}
SPL {X  -159.990, Y  +547.268, Z    +0.000, E1   +73.735, E3 +89200.449}
SPL {X  -159.091, Y  +360.560, Z    +0.000, E1   +74.726, E3 +89286.775}
SPL {X  -156.418, Y  +343.879, Z    +0.000, E1   +74.473, E3 +89299.201}
SPL {X  -153.414, Y  +332.103, Z    +0.000, E1   +74.378, E3 +89306.875}
SPL {X  -141.909, Y  +303.617, Z    +0.000, E1   +76.515, E3 +89299.405}
ENDSPLINE

SPLINE
SPL {X  -142.567, Y  +304.895, Z    +0.000, E1   +75.566, E3 +89308.220}
ENDSPLINE

SPLINE
SPL {X  -141.999, Y  +303.790, Z    +0.000, E1   +74.633, E3 +89317.472}
SPL {X  -141.780, Y  +303.371, Z    +0.000, E1   +73.549, E3 +89327.045}
SPL {X  -140.619, Y  +301.190, Z    +0.000, E1   +72.741, E3 +89334.892}
SPL {X  -137.438, Y  +295.601, Z    +0.000, E1   +72.365, E3 +89340.980}
SPL {X  -134.156, Y  +290.328, Z    +0.000, E1   +71.962, E3 +89346.851}
SPL {X  -130.677, Y  +285.194, Z    +0.000, E1   +71.519, E3 +89352.656}
SPL {X  -127.147, Y  +280.390, Z    +0.000, E1   +71.042, E3 +89358.140}
SPL {X  -123.431, Y  +275.709, Z    +0.000, E1   +70.518, E3 +89363.463}
SPL {X  -120.392, Y  +272.131, Z    +0.000, E1   +70.053, E3 +89367.484}
SPL {X   -79.311, Y  +238.552, Z    +0.000, E1   +58.563, E3 +89462.723}
ENDSPLINE

SPLINE
SPL {X  -105.077, Y  +256.854, Z    +0.000, E1   +55.187, E3 +89650.275}
SPL {X  -133.208, Y  +288.886, Z    +0.000, E1   +52.003, E3 +89683.376}
SPL {X  -149.825, Y  +321.381, Z    +0.000, E1   +42.580, E3 +89696.530}
SPL {X  -157.376, Y  +348.695, Z    +0.000, E1   +27.651, E3 +89701.615}
SPL {X  -159.486, Y  +364.808, Z    +0.000, E1   +14.693, E3 +89703.118}
SPL {X  -159.964, Y  +374.630, Z    +0.000, E1    +5.249, E3 +89703.523}
SPL {X  -159.990, Y  +379.484, Z    +0.000, E1    +0.034, E3 +89703.579}
SPL {X  -159.990, Y  +381.639, Z    +0.000, E1    -4.454, E3 +89703.601}
SPL {X  -159.990, Y  +387.459, Z    +0.000, E1   -18.927, E3 +89703.797}
SPL {X  -159.990, Y  +393.138, Z    +0.000, E1   -33.246, E3 +89704.146}
SPL {X  -159.990, Y  +399.326, Z    +0.000, E1   -44.934, E3 +89704.788}
SPL {X  -159.990, Y  +408.817, Z    +0.000, E1   -56.572, E3 +89706.161}
SPL {X  -159.990, Y  +426.617, Z    +0.000, E1   -66.230, E3 +89710.016}
SPL {X  -159.990, Y  +499.521, Z    +0.000, E1   -73.662, E3 +89733.343}
SPL {X  -159.629, Y  +687.249, Z    +0.000, E1   -74.539, E3 +89821.227}
SPL {X  -157.983, Y  +701.765, Z    +0.000, E1   -74.384, E3 +89831.459}
SPL {X  -155.520, Y  +714.054, Z    +0.000, E1   -74.151, E3 +89841.213}
SPL {X  -152.569, Y  +724.660, Z    +0.000, E1   -73.857, E3 +89850.448}
SPL {X  -149.625, Y  +733.149, Z    +0.000, E1   -73.553, E3 +89858.383}
SPL {X  -146.617, Y  +740.532, Z    +0.000, E1   -73.233, E3 +89865.659}
SPL {X  -143.394, Y  +747.457, Z    +0.000, E1   -72.883, E3 +89872.756}
SPL {X  -140.332, Y  +753.336, Z    +0.000, E1   -72.527, E3 +89879.031}
SPL {X  -137.187, Y  +758.820, Z    +0.000, E1   -72.156, E3 +89885.034}
SPL {X  -134.014, Y  +763.891, Z    +0.000, E1   -71.759, E3 +89890.720}
SPL {X  -130.657, Y  +768.834, Z    +0.000, E1   -71.330, E3 +89896.335}
SPL {X  -126.020, Y  +775.068, Z    +0.000, E1   -70.718, E3 +89903.463}
SPL {X  -121.287, Y  +780.838, Z    +0.000, E1   -70.013, E3 +89910.036}
SPL {X   -75.772, Y  +817.409, Z    +0.000, E1   -56.226, E3 +90037.389}
ENDSPLINE

SPLINE
SPL {X  -124.054, Y  +777.532, Z    +0.000, E1   -54.436, E3 +90220.617}
SPL {X  -149.719, Y  +732.901, Z    +0.000, E1   -43.150, E3 +90241.431}
SPL {X  -158.004, Y  +701.630, Z    +0.000, E1   -25.366, E3 +90246.896}
SPL {X  -159.838, Y  +683.473, Z    +0.000, E1    -9.532, E3 +90248.202}
SPL {X  -159.990, Y  +674.579, Z    +0.000, E1    -0.168, E3 +90248.385}
SPL {X  -159.990, Y  +672.677, Z    +0.000, E1    +3.879, E3 +90248.401}
SPL {X  -159.990, Y  +669.117, Z    +0.000, E1   +12.900, E3 +90248.483}
SPL {X  -159.990, Y  +663.639, Z    +0.000, E1   +26.675, E3 +90248.769}
SPL {X  -159.990, Y  +656.057, Z    +0.000, E1   +43.288, E3 +90249.425}
SPL {X  -159.990, Y  +647.797, Z    +0.000, E1   +54.469, E3 +90250.562}
SPL {X  -159.990, Y  +630.178, Z    +0.000, E1   +65.480, E3 +90254.246}
SPL {X  -159.990, Y  +547.268, Z    +0.000, E1   +73.735, E3 +90281.530}
SPL {X  -159.626, Y  +366.721, Z    +0.000, E1   +74.756, E3 +90363.795}
SPL {X  -158.582, Y  +356.317, Z    +0.000, E1   +74.662, E3 +90370.888}
SPL {X  -156.418, Y  +343.879, Z    +0.000, E1   +74.473, E3 +90380.282}
SPL {X  -153.414, Y  +332.103, Z    +0.000, E1   +74.378, E3 +90387.956}
SPL {X  -141.909, Y  +303.617, Z    +0.000, E1   +76.515, E3 +90380.486}
ENDSPLINE

SPLINE
SPL {X  -142.567, Y  +304.895, Z    +0.000, E1   +75.566, E3 +90389.301}
ENDSPLINE

SPLINE
SPL {X  -141.999, Y  +303.790, Z    +0.000, E1   +74.633, E3 +90398.553}
SPL {X  -141.780, Y  +303.371, Z    +0.000, E1   +73.549, E3 +90408.126}
SPL {X  -140.619, Y  +301.190, Z    +0.000, E1   +72.741, E3 +90415.973}
SPL {X  -137.438, Y  +295.601, Z    +0.000, E1   +72.365, E3 +90422.061}
SPL {X  -134.156, Y  +290.328, Z    +0.000, E1   +71.962, E3 +90427.932}
SPL {X  -130.677, Y  +285.194, Z    +0.000, E1   +71.519, E3 +90433.737}
SPL {X  -127.147, Y  +280.390, Z    +0.000, E1   +71.042, E3 +90439.221}
SPL {X  -123.431, Y  +275.709, Z    +0.000, E1   +70.518, E3 +90444.545}
SPL {X  -120.392, Y  +272.131, Z    +0.000, E1   +70.053, E3 +90448.565}
SPL {X   -79.311, Y  +238.552, Z    +0.000, E1   +58.563, E3 +90543.804}
ENDSPLINE

SPLINE
SPL {X  -105.077, Y  +256.854, Z    +0.000, E1   +55.187, E3 +90731.356}
SPL {X  -133.208, Y  +288.886, Z    +0.000, E1   +52.003, E3 +90764.457}
SPL {X  -149.825, Y  +321.381, Z    +0.000, E1   +42.580, E3 +90777.611}
SPL {X  -157.376, Y  +348.695, Z    +0.000, E1   +27.651, E3 +90782.696}
SPL {X  -159.486, Y  +364.808, Z    +0.000, E1   +14.693, E3 +90784.199}
SPL {X  -159.964, Y  +374.630, Z    +0.000, E1    +5.249, E3 +90784.604}
SPL {X  -159.990, Y  +379.484, Z    +0.000, E1    +0.034, E3 +90784.660}
SPL {X  -159.990, Y  +381.639, Z    +0.000, E1    -4.454, E3 +90784.682}
SPL {X  -159.990, Y  +385.871, Z    +0.000, E1   -15.161, E3 +90784.798}
SPL {X  -159.990, Y  +391.065, Z    +0.000, E1   -28.187, E3 +90785.086}
SPL {X  -159.990, Y  +399.326, Z    +0.000, E1   -44.934, E3 +90785.869}
SPL {X  -159.990, Y  +408.817, Z    +0.000, E1   -56.572, E3 +90787.242}
SPL {X  -159.990, Y  +426.617, Z    +0.000, E1   -66.230, E3 +90791.097}
SPL {X  -159.990, Y  +499.521, Z    +0.000, E1   -73.662, E3 +90814.424}
SPL {X  -159.629, Y  +687.249, Z    +0.000, E1   -74.539, E3 +90902.308}
SPL {X  -157.983, Y  +701.765, Z    +0.000, E1   -74.384, E3 +90912.540}
SPL {X  -155.520, Y  +714.054, Z    +0.000, E1   -74.151, E3 +90922.294}
SPL {X  -152.569, Y  +724.660, Z    +0.000, E1   -73.857, E3 +90931.529}
SPL {X  -149.625, Y  +733.149, Z    +0.000, E1   -73.553, E3 +90939.464}
SPL {X  -146.617, Y  +740.532, Z    +0.000, E1   -73.233, E3 +90946.740}
SPL {X  -143.394, Y  +747.457, Z    +0.000, E1   -72.883, E3 +90953.837}
SPL {X  -140.332, Y  +753.336, Z    +0.000, E1   -72.527, E3 +90960.112}
SPL {X  -137.187, Y  +758.820, Z    +0.000, E1   -72.156, E3 +90966.115}
SPL {X  -134.014, Y  +763.891, Z    +0.000, E1   -71.759, E3 +90971.801}
SPL {X  -130.657, Y  +768.834, Z    +0.000, E1   -71.330, E3 +90977.416}
SPL {X  -126.020, Y  +775.068, Z    +0.000, E1   -70.718, E3 +90984.544}
SPL {X  -121.287, Y  +780.838, Z    +0.000, E1   -70.013, E3 +90991.118}
SPL {X   -75.772, Y  +817.409, Z    +0.000, E1   -56.226, E3 +91118.470}
ENDSPLINE

SPLINE
SPL {X  -124.054, Y  +777.532, Z    +0.000, E1   -54.436, E3 +91301.698}
SPL {X  -149.719, Y  +732.901, Z    +0.000, E1   -43.150, E3 +91322.512}
SPL {X  -158.004, Y  +701.630, Z    +0.000, E1   -25.366, E3 +91327.977}
SPL {X  -159.639, Y  +687.095, Z    +0.000, E1   -12.931, E3 +91329.135}
SPL {X  -159.981, Y  +678.202, Z    +0.000, E1    -4.129, E3 +91329.429}
SPL {X  -159.990, Y  +674.500, Z    +0.000, E1    +0.000, E3 +91329.466}
SPL {X  -159.990, Y  +672.677, Z    +0.000, E1    +3.879, E3 +91329.482}
SPL {X  -159.990, Y  +669.117, Z    +0.000, E1   +12.900, E3 +91329.564}
SPL {X  -159.990, Y  +665.253, Z    +0.000, E1   +22.908, E3 +91329.738}
SPL {X  -159.990, Y  +658.335, Z    +0.000, E1   +38.839, E3 +91330.283}
SPL {X  -159.990, Y  +645.786, Z    +0.000, E1   +56.338, E3 +91331.997}
SPL {X  -159.990, Y  +623.264, Z    +0.000, E1   +67.753, E3 +91336.923}
SPL {X  -159.990, Y  +547.268, Z    +0.000, E1   +73.735, E3 +91362.611}
SPL {X  -159.626, Y  +366.721, Z    +0.000, E1   +74.756, E3 +91444.876}
SPL {X  -157.975, Y  +352.185, Z    +0.000, E1   +74.622, E3 +91454.942}
SPL {X  -154.546, Y  +336.120, Z    +0.000, E1   +74.400, E3 +91466.601}
SPL {X  -141.909, Y  +303.617, Z    +0.000, E1   +76.515, E3 +91461.567}
ENDSPLINE

SPLINE
SPL {X  -142.567, Y  +304.895, Z    +0.000, E1   +75.566, E3 +91470.383}
ENDSPLINE

SPLINE
SPL {X  -141.999, Y  +303.790, Z    +0.000, E1   +74.633, E3 +91479.634}
SPL {X  -141.780, Y  +303.371, Z    +0.000, E1   +73.549, E3 +91489.207}
SPL {X  -140.619, Y  +301.190, Z    +0.000, E1   +72.741, E3 +91497.054}
SPL {X  -137.438, Y  +295.601, Z    +0.000, E1   +72.365, E3 +91503.142}
SPL {X  -134.156, Y  +290.328, Z    +0.000, E1   +71.962, E3 +91509.013}
SPL {X  -130.677, Y  +285.194, Z    +0.000, E1   +71.519, E3 +91514.819}
SPL {X  -127.147, Y  +280.390, Z    +0.000, E1   +71.042, E3 +91520.303}
SPL {X  -123.431, Y  +275.709, Z    +0.000, E1   +70.518, E3 +91525.626}
SPL {X  -120.392, Y  +272.131, Z    +0.000, E1   +70.053, E3 +91529.646}
SPL {X   -79.311, Y  +238.552, Z    +0.000, E1   +58.563, E3 +91624.885}
ENDSPLINE

SPLINE
SPL {X  -105.077, Y  +256.854, Z    +0.000, E1   +55.187, E3 +91812.437}
SPL {X  -133.208, Y  +288.886, Z    +0.000, E1   +52.003, E3 +91845.538}
SPL {X  -149.825, Y  +321.381, Z    +0.000, E1   +42.580, E3 +91858.692}
SPL {X  -156.491, Y  +344.222, Z    +0.000, E1   +30.612, E3 +91863.198}
SPL {X  -159.275, Y  +362.387, Z    +0.000, E1   +16.907, E3 +91865.112}
SPL {X  -159.964, Y  +374.630, Z    +0.000, E1    +5.249, E3 +91865.685}
SPL {X  -159.990, Y  +379.735, Z    +0.000, E1    -0.236, E3 +91865.743}
SPL {X  -159.990, Y  +382.878, Z    +0.000, E1    -7.664, E3 +91865.782}
SPL {X  -159.990, Y  +387.459, Z    +0.000, E1   -18.927, E3 +91865.959}
SPL {X  -159.990, Y  +395.361, Z    +0.000, E1   -37.740, E3 +91866.523}
SPL {X  -159.990, Y  +406.369, Z    +0.000, E1   -54.148, E3 +91867.928}
SPL {X  -159.990, Y  +426.617, Z    +0.000, E1   -66.230, E3 +91872.178}
SPL {X  -159.990, Y  +499.521, Z    +0.000, E1   -73.662, E3 +91895.505}
SPL {X  -159.629, Y  +687.249, Z    +0.000, E1   -74.539, E3 +91983.389}
SPL {X  -157.983, Y  +701.765, Z    +0.000, E1   -74.384, E3 +91993.621}
SPL {X  -155.520, Y  +714.054, Z    +0.000, E1   -74.151, E3 +92003.375}
SPL {X  -152.569, Y  +724.660, Z    +0.000, E1   -73.857, E3 +92012.610}
SPL {X  -149.625, Y  +733.149, Z    +0.000, E1   -73.553, E3 +92020.545}
SPL {X  -146.617, Y  +740.532, Z    +0.000, E1   -73.233, E3 +92027.821}
SPL {X  -143.394, Y  +747.457, Z    +0.000, E1   -72.883, E3 +92034.918}
SPL {X  -140.332, Y  +753.336, Z    +0.000, E1   -72.527, E3 +92041.193}
SPL {X  -137.187, Y  +758.820, Z    +0.000, E1   -72.156, E3 +92047.196}
SPL {X  -134.014, Y  +763.891, Z    +0.000, E1   -71.759, E3 +92052.882}
SPL {X  -129.643, Y  +770.252, Z    +0.000, E1   -71.218, E3 +92060.089}
SPL {X  -125.230, Y  +776.071, Z    +0.000, E1   -70.580, E3 +92066.807}
SPL {X  -121.287, Y  +780.838, Z    +0.000, E1   -70.013, E3 +92072.199}
SPL {X   -75.772, Y  +817.409, Z    +0.000, E1   -56.226, E3 +92199.551}
ENDSPLINE

SPLINE
SPL {X  -124.054, Y  +777.532, Z    +0.000, E1   -54.436, E3 +92382.779}
SPL {X  -145.922, Y  +742.101, Z    +0.000, E1   -46.535, E3 +92401.048}
SPL {X  -155.216, Y  +715.293, Z    +0.000, E1   -34.460, E3 +92407.241}
SPL {X  -158.715, Y  +696.660, Z    +0.000, E1   -21.368, E3 +92409.568}
SPL {X  -159.838, Y  +683.473, Z    +0.000, E1    -9.532, E3 +92410.364}
SPL {X  -159.990, Y  +674.579, Z    +0.000, E1    -0.168, E3 +92410.547}
SPL {X  -159.990, Y  +672.677, Z    +0.000, E1    +3.879, E3 +92410.563}
SPL {X  -159.990, Y  +669.117, Z    +0.000, E1   +12.900, E3 +92410.645}
SPL {X  -159.990, Y  +665.253, Z    +0.000, E1   +22.908, E3 +92410.819}
SPL {X  -159.990, Y  +658.335, Z    +0.000, E1   +38.839, E3 +92411.364}
SPL {X  -159.990, Y  +647.797, Z    +0.000, E1   +54.469, E3 +92412.724}
SPL {X  -159.990, Y  +630.178, Z    +0.000, E1   +65.480, E3 +92416.408}
SPL {X  -159.990, Y  +547.268, Z    +0.000, E1   +73.735, E3 +92443.692}
SPL {X  -159.091, Y  +360.560, Z    +0.000, E1   +74.726, E3 +92530.018}
SPL {X  -156.418, Y  +343.879, Z    +0.000, E1   +74.473, E3 +92542.444}
SPL {X  -153.414, Y  +332.103, Z    +0.000, E1   +74.378, E3 +92550.119}
SPL {X  -141.909, Y  +303.617, Z    +0.000, E1   +76.515, E3 +92542.649}
ENDSPLINE

SPLINE
SPL {X  -142.567, Y  +304.895, Z    +0.000, E1   +75.566, E3 +92551.464}
ENDSPLINE

SPLINE
SPL {X  -141.999, Y  +303.790, Z    +0.000, E1   +74.633, E3 +92560.715}
SPL {X  -141.780, Y  +303.371, Z    +0.000, E1   +73.549, E3 +92570.289}
SPL {X  -140.619, Y  +301.190, Z    +0.000, E1   +72.741, E3 +92578.135}
SPL {X  -137.438, Y  +295.601, Z    +0.000, E1   +72.365, E3 +92584.223}
SPL {X  -134.156, Y  +290.328, Z    +0.000, E1   +71.962, E3 +92590.095}
SPL {X  -130.677, Y  +285.194, Z    +0.000, E1   +71.519, E3 +92595.900}
SPL {X  -126.239, Y  +279.212, Z    +0.000, E1   +70.937, E3 +92602.701}
SPL {X  -121.335, Y  +273.218, Z    +0.000, E1   +70.225, E3 +92609.489}
SPL {X   -79.311, Y  +238.552, Z    +0.000, E1   +58.563, E3 +92705.966}
ENDSPLINE

SPLINE
SPL {X  -105.077, Y  +256.854, Z    +0.000, E1   +55.187, E3 +92893.518}
SPL {X  -133.208, Y  +288.886, Z    +0.000, E1   +52.003, E3 +92926.620}
SPL {X  -149.825, Y  +321.381, Z    +0.000, E1   +42.580, E3 +92939.773}
SPL {X  -157.376, Y  +348.695, Z    +0.000, E1   +27.651, E3 +92944.858}
SPL {X  -159.486, Y  +364.808, Z    +0.000, E1   +14.693, E3 +92946.361}
SPL {X  -159.964, Y  +374.630, Z    +0.000, E1    +5.249, E3 +92946.766}
SPL {X  -159.990, Y  +379.484, Z    +0.000, E1    +0.034, E3 +92946.822}
SPL {X  -159.990, Y  +381.639, Z    +0.000, E1    -4.454, E3 +92946.844}
SPL {X  -159.990, Y  +387.459, Z    +0.000, E1   -18.927, E3 +92947.040}
SPL {X  -159.990, Y  +393.138, Z    +0.000, E1   -33.246, E3 +92947.389}
SPL {X  -159.990, Y  +399.326, Z    +0.000, E1   -44.934, E3 +92948.031}
SPL {X  -159.990, Y  +408.817, Z    +0.000, E1   -56.572, E3 +92949.404}
SPL {X  -159.990, Y  +426.617, Z    +0.000, E1   -66.230, E3 +92953.259}
SPL {X  -159.990, Y  +499.521, Z    +0.000, E1   -73.662, E3 +92976.586}
SPL {X  -159.629, Y  +687.249, Z    +0.000, E1   -74.539, E3 +93064.470}
SPL {X  -157.983, Y  +701.765, Z    +0.000, E1   -74.384, E3 +93074.702}
SPL {X  -155.520, Y  +714.054, Z    +0.000, E1   -74.151, E3 +93084.456}
SPL {X  -152.569, Y  +724.660, Z    +0.000, E1   -73.857, E3 +93093.691}
SPL {X  -149.625, Y  +733.149, Z    +0.000, E1   -73.553, E3 +93101.626}
SPL {X  -146.617, Y  +740.532, Z    +0.000, E1   -73.233, E3 +93108.903}
SPL {X  -143.394, Y  +747.457, Z    +0.000, E1   -72.883, E3 +93115.999}
SPL {X  -140.332, Y  +753.336, Z    +0.000, E1   -72.527, E3 +93122.274}
SPL {X  -137.187, Y  +758.820, Z    +0.000, E1   -72.156, E3 +93128.277}
SPL {X  -134.014, Y  +763.891, Z    +0.000, E1   -71.759, E3 +93133.963}
SPL {X  -129.643, Y  +770.252, Z    +0.000, E1   -71.218, E3 +93141.170}
SPL {X  -125.230, Y  +776.071, Z    +0.000, E1   -70.580, E3 +93147.888}
SPL {X  -122.263, Y  +779.692, Z    +0.000, E1   -70.136, E3 +93152.018}
SPL {X  -120.205, Y  +782.082, Z    +0.000, E1   -69.822, E3 +93154.693}
SPL {X   -77.717, Y  +816.346, Z    +0.000, E1   -57.422, E3 +93262.544}
SPL {X   -74.440, Y  +818.117, Z    +0.000, E1   -54.647, E3 +93315.784}
ENDSPLINE

SPLINE
SPL {X  -124.054, Y  +777.532, Z    +0.000, E1   -54.436, E3 +93463.860}
SPL {X  -149.719, Y  +732.901, Z    +0.000, E1   -43.150, E3 +93484.674}
SPL {X  -158.004, Y  +701.630, Z    +0.000, E1   -25.366, E3 +93490.139}
SPL {X  -159.838, Y  +683.473, Z    +0.000, E1    -9.532, E3 +93491.445}
SPL {X  -159.990, Y  +674.579, Z    +0.000, E1    -0.168, E3 +93491.628}
SPL {X  -159.990, Y  +672.677, Z    +0.000, E1    +3.879, E3 +93491.644}
SPL {X  -159.990, Y  +669.117, Z    +0.000, E1   +12.900, E3 +93491.726}
SPL {X  -159.990, Y  +665.253, Z    +0.000, E1   +22.908, E3 +93491.900}
SPL {X  -159.990, Y  +658.335, Z    +0.000, E1   +38.839, E3 +93492.445}
SPL {X  -159.990, Y  +647.797, Z    +0.000, E1   +54.469, E3 +93493.805}
SPL {X  -159.990, Y  +630.178, Z    +0.000, E1   +65.480, E3 +93497.489}
SPL {X  -159.990, Y  +547.268, Z    +0.000, E1   +73.735, E3 +93524.773}
SPL {X  -159.091, Y  +360.560, Z    +0.000, E1   +74.726, E3 +93611.099}
SPL {X  -156.418, Y  +343.879, Z    +0.000, E1   +74.473, E3 +93623.525}
SPL {X  -153.414, Y  +332.103, Z    +0.000, E1   +74.378, E3 +93631.200}
SPL {X  -141.909, Y  +303.617, Z    +0.000, E1   +76.515, E3 +93623.730}
ENDSPLINE

SPLINE
SPL {X  -142.567, Y  +304.895, Z    +0.000, E1   +75.566, E3 +93632.545}
ENDSPLINE

SPLINE
SPL {X  -141.999, Y  +303.790, Z    +0.000, E1   +74.633, E3 +93641.796}
SPL {X  -141.780, Y  +303.371, Z    +0.000, E1   +73.549, E3 +93651.370}
SPL {X  -140.619, Y  +301.190, Z    +0.000, E1   +72.741, E3 +93659.216}
SPL {X  -137.438, Y  +295.601, Z    +0.000, E1   +72.365, E3 +93665.305}
SPL {X  -134.156, Y  +290.328, Z    +0.000, E1   +71.962, E3 +93671.176}
SPL {X  -130.677, Y  +285.194, Z    +0.000, E1   +71.519, E3 +93676.981}
SPL {X  -127.147, Y  +280.390, Z    +0.000, E1   +71.042, E3 +93682.465}
SPL {X  -123.431, Y  +275.709, Z    +0.000, E1   +70.518, E3 +93687.788}
SPL {X  -120.392, Y  +272.131, Z    +0.000, E1   +70.053, E3 +93691.808}
SPL {X   -79.311, Y  +238.552, Z    +0.000, E1   +58.563, E3 +93787.047}
ENDSPLINE

SPLINE
SPL {X  -105.077, Y  +256.854, Z    +0.000, E1   +55.187, E3 +93974.600}
SPL {X  -133.208, Y  +288.886, Z    +0.000, E1   +52.003, E3 +94007.701}
SPL {X  -149.825, Y  +321.381, Z    +0.000, E1   +42.580, E3 +94020.854}
SPL {X  -156.491, Y  +344.222, Z    +0.000, E1   +30.612, E3 +94025.360}
SPL {X  -159.275, Y  +362.387, Z    +0.000, E1   +16.907, E3 +94027.274}
SPL {X  -159.964, Y  +374.630, Z    +0.000, E1    +5.249, E3 +94027.848}
SPL {X  -159.990, Y  +379.484, Z    +0.000, E1    +0.034, E3 +94027.903}
SPL {X  -159.990, Y  +381.639, Z    +0.000, E1    -4.454, E3 +94027.925}
SPL {X  -159.990, Y  +385.871, Z    +0.000, E1   -15.161, E3 +94028.041}
SPL {X  -159.990, Y  +391.065, Z    +0.000, E1   -28.187, E3 +94028.329}
SPL {X  -159.990, Y  +397.286, Z    +0.000, E1   -41.591, E3 +94028.872}
SPL {X  -159.990, Y  +406.369, Z    +0.000, E1   -54.148, E3 +94030.091}
SPL {X  -159.990, Y  +426.617, Z    +0.000, E1   -66.230, E3 +94034.340}
SPL {X  -159.990, Y  +499.521, Z    +0.000, E1   -73.662, E3 +94057.667}
SPL {X  -159.629, Y  +687.249, Z    +0.000, E1   -74.539, E3 +94145.551}
SPL {X  -157.983, Y  +701.765, Z    +0.000, E1   -74.384, E3 +94155.783}
SPL {X  -155.520, Y  +714.054, Z    +0.000, E1   -74.151, E3 +94165.537}
SPL {X  -152.569, Y  +724.660, Z    +0.000, E1   -73.857, E3 +94174.772}
SPL {X  -149.625, Y  +733.149, Z    +0.000, E1   -73.553, E3 +94182.707}
SPL {X  -146.617, Y  +740.532, Z    +0.000, E1   -73.233, E3 +94189.984}
SPL {X  -143.394, Y  +747.457, Z    +0.000, E1   -72.883, E3 +94197.081}
SPL {X  -140.332, Y  +753.336, Z    +0.000, E1   -72.527, E3 +94203.356}
SPL {X  -137.187, Y  +758.820, Z    +0.000, E1   -72.156, E3 +94209.359}
SPL {X  -134.014, Y  +763.891, Z    +0.000, E1   -71.759, E3 +94215.044}
SPL {X  -130.657, Y  +768.834, Z    +0.000, E1   -71.330, E3 +94220.659}
SPL {X  -126.020, Y  +775.068, Z    +0.000, E1   -70.718, E3 +94227.787}
SPL {X  -121.287, Y  +780.838, Z    +0.000, E1   -70.013, E3 +94234.361}
SPL {X   -75.772, Y  +817.409, Z    +0.000, E1   -56.226, E3 +94361.713}
ENDSPLINE

SPLINE
SPL {X  -124.054, Y  +777.532, Z    +0.000, E1   -54.436, E3 +94544.941}
SPL {X  -145.922, Y  +742.101, Z    +0.000, E1   -46.535, E3 +94563.211}
SPL {X  -155.216, Y  +715.293, Z    +0.000, E1   -34.460, E3 +94569.403}
SPL {X  -158.715, Y  +696.660, Z    +0.000, E1   -21.368, E3 +94571.731}
SPL {X  -159.838, Y  +683.473, Z    +0.000, E1    -9.532, E3 +94572.526}
SPL {X  -159.990, Y  +674.579, Z    +0.000, E1    -0.168, E3 +94572.709}
SPL {X  -159.990, Y  +672.677, Z    +0.000, E1    +3.879, E3 +94572.725}
SPL {X  -159.990, Y  +669.117, Z    +0.000, E1   +12.900, E3 +94572.808}
SPL {X  -159.990, Y  +663.639, Z    +0.000, E1   +26.675, E3 +94573.093}
SPL {X  -159.990, Y  +656.057, Z    +0.000, E1   +43.288, E3 +94573.749}
SPL {X  -159.990, Y  +647.797, Z    +0.000, E1   +54.469, E3 +94574.886}
SPL {X  -159.990, Y  +630.178, Z    +0.000, E1   +65.480, E3 +94578.570}
SPL {X  -159.990, Y  +547.268, Z    +0.000, E1   +73.735, E3 +94605.854}
SPL {X  -159.091, Y  +360.560, Z    +0.000, E1   +74.726, E3 +94692.181}
SPL {X  -156.418, Y  +343.879, Z    +0.000, E1   +74.473, E3 +94704.606}
SPL {X  -153.414, Y  +332.103, Z    +0.000, E1   +74.378, E3 +94712.281}
SPL {X  -141.909, Y  +303.617, Z    +0.000, E1   +76.515, E3 +94704.811}
ENDSPLINE

SPLINE
SPL {X  -142.567, Y  +304.895, Z    +0.000, E1   +75.566, E3 +94713.626}
ENDSPLINE

SPLINE
SPL {X  -141.999, Y  +303.790, Z    +0.000, E1   +74.633, E3 +94722.877}
SPL {X  -141.780, Y  +303.371, Z    +0.000, E1   +73.549, E3 +94732.451}
SPL {X  -140.619, Y  +301.190, Z    +0.000, E1   +72.741, E3 +94740.297}
SPL {X  -137.438, Y  +295.601, Z    +0.000, E1   +72.365, E3 +94746.386}
SPL {X  -134.156, Y  +290.328, Z    +0.000, E1   +71.962, E3 +94752.257}
SPL {X  -130.677, Y  +285.194, Z    +0.000, E1   +71.519, E3 +94758.062}
SPL {X  -127.147, Y  +280.390, Z    +0.000, E1   +71.042, E3 +94763.546}
SPL {X  -123.431, Y  +275.709, Z    +0.000, E1   +70.518, E3 +94768.869}
SPL {X  -120.392, Y  +272.131, Z    +0.000, E1   +70.053, E3 +94772.889}
SPL {X   -79.311, Y  +238.552, Z    +0.000, E1   +58.563, E3 +94868.128}
ENDSPLINE

SPLINE
SPL {X  -105.077, Y  +256.854, Z    +0.000, E1   +55.187, E3 +95055.681}
SPL {X  -133.208, Y  +288.886, Z    +0.000, E1   +52.003, E3 +95088.782}
SPL {X  -149.825, Y  +321.381, Z    +0.000, E1   +42.580, E3 +95101.935}
SPL {X  -157.376, Y  +348.695, Z    +0.000, E1   +27.651, E3 +95107.020}
SPL {X  -159.486, Y  +364.808, Z    +0.000, E1   +14.693, E3 +95108.523}
SPL {X  -159.964, Y  +374.630, Z    +0.000, E1    +5.249, E3 +95108.929}
SPL {X  -159.990, Y  +379.735, Z    +0.000, E1    -0.236, E3 +95108.986}
SPL {X  -159.990, Y  +384.648, Z    +0.000, E1   -11.739, E3 +95109.082}
SPL {X  -159.990, Y  +391.065, Z    +0.000, E1   -28.187, E3 +95109.410}
SPL {X  -159.990, Y  +399.326, Z    +0.000, E1   -44.934, E3 +95110.193}
SPL {X  -159.990, Y  +408.817, Z    +0.000, E1   -56.572, E3 +95111.566}
SPL {X  -159.990, Y  +426.617, Z    +0.000, E1   -66.230, E3 +95115.421}
SPL {X  -159.990, Y  +499.521, Z    +0.000, E1   -73.662, E3 +95138.748}
SPL {X  -159.629, Y  +687.249, Z    +0.000, E1   -74.539, E3 +95226.632}
SPL {X  -157.983, Y  +701.765, Z    +0.000, E1   -74.384, E3 +95236.864}
SPL {X  -155.520, Y  +714.054, Z    +0.000, E1   -74.151, E3 +95246.619}
SPL {X  -152.569, Y  +724.660, Z    +0.000, E1   -73.857, E3 +95255.853}
SPL {X  -149.625, Y  +733.149, Z    +0.000, E1   -73.553, E3 +95263.788}
SPL {X  -146.617, Y  +740.532, Z    +0.000, E1   -73.233, E3 +95271.065}
SPL {X  -143.394, Y  +747.457, Z    +0.000, E1   -72.883, E3 +95278.162}
SPL {X  -140.332, Y  +753.336, Z    +0.000, E1   -72.527, E3 +95284.437}
SPL {X  -137.187, Y  +758.820, Z    +0.000, E1   -72.156, E3 +95290.440}
SPL {X  -134.014, Y  +763.891, Z    +0.000, E1   -71.759, E3 +95296.125}
SPL {X  -130.657, Y  +768.834, Z    +0.000, E1   -71.330, E3 +95301.741}
SPL {X  -126.937, Y  +773.885, Z    +0.000, E1   -70.823, E3 +95307.542}
SPL {X  -122.983, Y  +778.833, Z    +0.000, E1   -70.262, E3 +95313.187}
SPL {X  -120.205, Y  +782.082, Z    +0.000, E1   -69.822, E3 +95316.855}
SPL {X   -77.717, Y  +816.346, Z    +0.000, E1   -57.422, E3 +95424.707}
SPL {X   -74.440, Y  +818.117, Z    +0.000, E1   -54.647, E3 +95477.946}
ENDSPLINE

SPLINE
SPL {X  -124.054, Y  +777.532, Z    +0.000, E1   -54.436, E3 +95626.022}
SPL {X  -149.719, Y  +732.901, Z    +0.000, E1   -43.150, E3 +95646.836}
SPL {X  -158.004, Y  +701.630, Z    +0.000, E1   -25.366, E3 +95652.301}
SPL {X  -159.838, Y  +683.473, Z    +0.000, E1    -9.532, E3 +95653.608}
SPL {X  -159.990, Y  +674.579, Z    +0.000, E1    -0.168, E3 +95653.790}
SPL {X  -159.990, Y  +672.677, Z    +0.000, E1    +3.879, E3 +95653.806}
SPL {X  -159.990, Y  +669.117, Z    +0.000, E1   +12.900, E3 +95653.889}
SPL {X  -159.990, Y  +665.253, Z    +0.000, E1   +22.908, E3 +95654.062}
SPL {X  -159.990, Y  +658.335, Z    +0.000, E1   +38.839, E3 +95654.607}
SPL {X  -159.990, Y  +645.786, Z    +0.000, E1   +56.338, E3 +95656.321}
SPL {X  -159.990, Y  +623.264, Z    +0.000, E1   +67.753, E3 +95661.247}
SPL {X  -159.990, Y  +547.268, Z    +0.000, E1   +73.735, E3 +95686.935}
SPL {X  -159.091, Y  +360.560, Z    +0.000, E1   +74.726, E3 +95773.262}
SPL {X  -156.418, Y  +343.879, Z    +0.000, E1   +74.473, E3 +95785.687}
SPL {X  -153.414, Y  +332.103, Z    +0.000, E1   +74.378, E3 +95793.362}
SPL {X  -141.909, Y  +303.617, Z    +0.000, E1   +76.515, E3 +95785.892}
ENDSPLINE

SPLINE
SPL {X  -142.567, Y  +304.895, Z    +0.000, E1   +75.566, E3 +95794.707}
ENDSPLINE

SPLINE
SPL {X  -141.999, Y  +303.790, Z    +0.000, E1   +74.633, E3 +95803.958}
SPL {X  -141.780, Y  +303.371, Z    +0.000, E1   +73.549, E3 +95813.532}
SPL {X  -140.619, Y  +301.190, Z    +0.000, E1   +72.741, E3 +95821.378}
SPL {X  -137.438, Y  +295.601, Z    +0.000, E1   +72.365, E3 +95827.467}
SPL {X  -134.156, Y  +290.328, Z    +0.000, E1   +71.962, E3 +95833.338}
SPL {X  -130.677, Y  +285.194, Z    +0.000, E1   +71.519, E3 +95839.143}
SPL {X  -127.147, Y  +280.390, Z    +0.000, E1   +71.042, E3 +95844.627}
SPL {X  -123.431, Y  +275.709, Z    +0.000, E1   +70.518, E3 +95849.950}
SPL {X  -120.392, Y  +272.131, Z    +0.000, E1   +70.053, E3 +95853.970}
SPL {X   -79.311, Y  +238.552, Z    +0.000, E1   +58.563, E3 +95949.209}
ENDSPLINE

SPLINE
SPL {X  -105.077, Y  +256.854, Z    +0.000, E1   +55.187, E3 +96136.762}
SPL {X  -133.208, Y  +288.886, Z    +0.000, E1   +52.003, E3 +96169.863}
SPL {X  -149.825, Y  +321.381, Z    +0.000, E1   +42.580, E3 +96183.016}
SPL {X  -157.376, Y  +348.695, Z    +0.000, E1   +27.651, E3 +96188.101}
SPL {X  -159.486, Y  +364.808, Z    +0.000, E1   +14.693, E3 +96189.604}
SPL {X  -159.964, Y  +374.630, Z    +0.000, E1    +5.249, E3 +96190.010}
SPL {X  -159.990, Y  +379.735, Z    +0.000, E1    -0.236, E3 +96190.067}
SPL {X  -159.990, Y  +384.648, Z    +0.000, E1   -11.739, E3 +96190.164}
SPL {X  -159.990, Y  +391.065, Z    +0.000, E1   -28.187, E3 +96190.491}
SPL {X  -159.990, Y  +399.326, Z    +0.000, E1   -44.934, E3 +96191.274}
SPL {X  -159.990, Y  +408.817, Z    +0.000, E1   -56.572, E3 +96192.647}
SPL {X  -159.990, Y  +426.617, Z    +0.000, E1   -66.230, E3 +96196.503}
SPL {X  -159.990, Y  +499.521, Z    +0.000, E1   -73.662, E3 +96219.829}
SPL {X  -159.629, Y  +687.249, Z    +0.000, E1   -74.539, E3 +96307.713}
SPL {X  -157.983, Y  +701.765, Z    +0.000, E1   -74.384, E3 +96317.946}
SPL {X  -155.520, Y  +714.054, Z    +0.000, E1   -74.151, E3 +96327.700}
SPL {X  -152.569, Y  +724.660, Z    +0.000, E1   -73.857, E3 +96336.934}
SPL {X  -149.625, Y  +733.149, Z    +0.000, E1   -73.553, E3 +96344.869}
SPL {X  -146.617, Y  +740.532, Z    +0.000, E1   -73.233, E3 +96352.146}
SPL {X  -143.394, Y  +747.457, Z    +0.000, E1   -72.883, E3 +96359.243}
SPL {X  -140.332, Y  +753.336, Z    +0.000, E1   -72.527, E3 +96365.518}
SPL {X  -137.187, Y  +758.820, Z    +0.000, E1   -72.156, E3 +96371.521}
SPL {X  -134.014, Y  +763.891, Z    +0.000, E1   -71.759, E3 +96377.206}
SPL {X  -130.657, Y  +768.834, Z    +0.000, E1   -71.330, E3 +96382.822}
SPL {X  -126.020, Y  +775.068, Z    +0.000, E1   -70.718, E3 +96389.949}
SPL {X  -121.287, Y  +780.838, Z    +0.000, E1   -70.013, E3 +96396.523}
SPL {X   -75.772, Y  +817.409, Z    +0.000, E1   -56.226, E3 +96523.875}
ENDSPLINE

SPLINE
SPL {X  -124.054, Y  +777.532, Z    +0.000, E1   -54.436, E3 +96707.103}
SPL {X  -149.719, Y  +732.901, Z    +0.000, E1   -43.150, E3 +96727.917}
SPL {X  -158.004, Y  +701.630, Z    +0.000, E1   -25.366, E3 +96733.382}
SPL {X  -159.639, Y  +687.095, Z    +0.000, E1   -12.931, E3 +96734.540}
SPL {X  -159.981, Y  +678.202, Z    +0.000, E1    -4.129, E3 +96734.834}
SPL {X  -159.990, Y  +674.500, Z    +0.000, E1    +0.000, E3 +96734.872}
SPL {X  -159.990, Y  +672.677, Z    +0.000, E1    +3.879, E3 +96734.887}
SPL {X  -159.990, Y  +669.117, Z    +0.000, E1   +12.900, E3 +96734.970}
SPL {X  -159.990, Y  +663.639, Z    +0.000, E1   +26.675, E3 +96735.255}
SPL {X  -159.990, Y  +656.057, Z    +0.000, E1   +43.288, E3 +96735.911}
SPL {X  -159.990, Y  +645.786, Z    +0.000, E1   +56.338, E3 +96737.402}
SPL {X  -159.990, Y  +623.264, Z    +0.000, E1   +67.753, E3 +96742.328}
SPL {X  -159.990, Y  +547.268, Z    +0.000, E1   +73.735, E3 +96768.016}
SPL {X  -159.091, Y  +360.560, Z    +0.000, E1   +74.726, E3 +96854.343}
SPL {X  -156.418, Y  +343.879, Z    +0.000, E1   +74.473, E3 +96866.768}
SPL {X  -153.414, Y  +332.103, Z    +0.000, E1   +74.378, E3 +96874.443}
SPL {X  -141.909, Y  +303.617, Z    +0.000, E1   +76.515, E3 +96866.973}
ENDSPLINE

SPLINE
SPL {X  -142.567, Y  +304.895, Z    +0.000, E1   +75.566, E3 +96875.788}
ENDSPLINE

SPLINE
SPL {X  -141.999, Y  +303.790, Z    +0.000, E1   +74.633, E3 +96885.039}
SPL {X  -141.780, Y  +303.371, Z    +0.000, E1   +73.549, E3 +96894.613}
SPL {X  -140.619, Y  +301.190, Z    +0.000, E1   +72.741, E3 +96902.460}
SPL {X  -137.438, Y  +295.601, Z    +0.000, E1   +72.365, E3 +96908.548}
SPL {X  -134.156, Y  +290.328, Z    +0.000, E1   +71.962, E3 +96914.419}
SPL {X  -130.677, Y  +285.194, Z    +0.000, E1   +71.519, E3 +96920.224}
SPL {X  -126.239, Y  +279.212, Z    +0.000, E1   +70.937, E3 +96927.025}
SPL {X  -121.335, Y  +273.218, Z    +0.000, E1   +70.225, E3 +96933.813}
SPL {X   -79.311, Y  +238.552, Z    +0.000, E1   +58.563, E3 +97030.290}
ENDSPLINE

SPLINE
SPL {X  -105.077, Y  +256.854, Z    +0.000, E1   +55.187, E3 +97217.843}
SPL {X  -133.208, Y  +288.886, Z    +0.000, E1   +52.003, E3 +97250.944}
SPL {X  -149.825, Y  +321.381, Z    +0.000, E1   +42.580, E3 +97264.097}
SPL {X  -156.491, Y  +344.222, Z    +0.000, E1   +30.612, E3 +97268.604}
SPL {X  -159.275, Y  +362.387, Z    +0.000, E1   +16.907, E3 +97270.517}
SPL {X  -159.964, Y  +374.630, Z    +0.000, E1    +5.249, E3 +97271.091}
SPL {X  -159.990, Y  +379.484, Z    +0.000, E1    +0.034, E3 +97271.147}
SPL {X  -159.990, Y  +381.639, Z    +0.000, E1    -4.454, E3 +97271.168}
SPL {X  -159.990, Y  +385.871, Z    +0.000, E1   -15.161, E3 +97271.284}
SPL {X  -159.990, Y  +391.065, Z    +0.000, E1   -28.187, E3 +97271.572}
SPL {X  -159.990, Y  +397.286, Z    +0.000, E1   -41.591, E3 +97272.115}
SPL {X  -159.990, Y  +406.369, Z    +0.000, E1   -54.148, E3 +97273.334}
SPL {X  -159.990, Y  +426.617, Z    +0.000, E1   -66.230, E3 +97277.584}
SPL {X  -159.990, Y  +499.521, Z    +0.000, E1   -73.662, E3 +97300.910}
SPL {X  -159.629, Y  +687.249, Z    +0.000, E1   -74.539, E3 +97388.794}
SPL {X  -157.983, Y  +701.765, Z    +0.000, E1   -74.384, E3 +97399.027}
SPL {X  -155.520, Y  +714.054, Z    +0.000, E1   -74.151, E3 +97408.781}
SPL {X  -152.569, Y  +724.660, Z    +0.000, E1   -73.857, E3 +97418.015}
SPL {X  -149.625, Y  +733.149, Z    +0.000, E1   -73.553, E3 +97425.950}
SPL {X  -146.617, Y  +740.532, Z    +0.000, E1   -73.233, E3 +97433.227}
SPL {X  -143.394, Y  +747.457, Z    +0.000, E1   -72.883, E3 +97440.324}
SPL {X  -140.332, Y  +753.336, Z    +0.000, E1   -72.527, E3 +97446.599}
SPL {X  -137.187, Y  +758.820, Z    +0.000, E1   -72.156, E3 +97452.602}
SPL {X  -134.014, Y  +763.891, Z    +0.000, E1   -71.759, E3 +97458.287}
SPL {X  -130.657, Y  +768.834, Z    +0.000, E1   -71.330, E3 +97463.903}
SPL {X  -126.020, Y  +775.068, Z    +0.000, E1   -70.718, E3 +97471.030}
SPL {X  -121.287, Y  +780.838, Z    +0.000, E1   -70.013, E3 +97477.604}
SPL {X   -75.772, Y  +817.409, Z    +0.000, E1   -56.226, E3 +97604.956}
ENDSPLINE

SPLINE
SPL {X  -124.054, Y  +777.532, Z    +0.000, E1   -54.436, E3 +97788.184}
SPL {X  -149.719, Y  +732.901, Z    +0.000, E1   -43.150, E3 +97808.998}
SPL {X  -158.004, Y  +701.630, Z    +0.000, E1   -25.366, E3 +97814.463}
SPL {X  -159.838, Y  +683.473, Z    +0.000, E1    -9.532, E3 +97815.770}
SPL {X  -159.990, Y  +674.579, Z    +0.000, E1    -0.168, E3 +97815.952}
SPL {X  -159.990, Y  +672.677, Z    +0.000, E1    +3.879, E3 +97815.968}
SPL {X  -159.990, Y  +669.117, Z    +0.000, E1   +12.900, E3 +97816.051}
SPL {X  -159.990, Y  +663.639, Z    +0.000, E1   +26.675, E3 +97816.336}
SPL {X  -159.990, Y  +656.057, Z    +0.000, E1   +43.288, E3 +97816.992}
SPL {X  -159.990, Y  +647.797, Z    +0.000, E1   +54.469, E3 +97818.129}
SPL {X  -159.990, Y  +630.178, Z    +0.000, E1   +65.480, E3 +97821.813}
SPL {X  -159.990, Y  +547.268, Z    +0.000, E1   +73.735, E3 +97849.097}
SPL {X  -159.626, Y  +366.721, Z    +0.000, E1   +74.756, E3 +97931.363}
SPL {X  -158.582, Y  +356.317, Z    +0.000, E1   +74.662, E3 +97938.456}
SPL {X  -156.418, Y  +343.879, Z    +0.000, E1   +74.473, E3 +97947.849}
SPL {X  -153.414, Y  +332.103, Z    +0.000, E1   +74.378, E3 +97955.524}
SPL {X  -141.909, Y  +303.617, Z    +0.000, E1   +76.515, E3 +97948.054}
ENDSPLINE

SPLINE
SPL {X  -142.567, Y  +304.895, Z    +0.000, E1   +75.566, E3 +97956.869}
ENDSPLINE

SPLINE
SPL {X  -141.999, Y  +303.790, Z    +0.000, E1   +74.633, E3 +97966.120}
SPL {X  -141.780, Y  +303.371, Z    +0.000, E1   +73.549, E3 +97975.694}
SPL {X  -140.619, Y  +301.190, Z    +0.000, E1   +72.741, E3 +97983.541}
SPL {X  -137.438, Y  +295.601, Z    +0.000, E1   +72.365, E3 +97989.629}
SPL {X  -134.156, Y  +290.328, Z    +0.000, E1   +71.962, E3 +97995.500}
SPL {X  -130.677, Y  +285.194, Z    +0.000, E1   +71.519, E3 +98001.305}
SPL {X  -127.147, Y  +280.390, Z    +0.000, E1   +71.042, E3 +98006.789}
SPL {X  -123.431, Y  +275.709, Z    +0.000, E1   +70.518, E3 +98012.112}
SPL {X  -120.392, Y  +272.131, Z    +0.000, E1   +70.053, E3 +98016.133}
SPL {X   -79.311, Y  +238.552, Z    +0.000, E1   +58.563, E3 +98111.371}
ENDSPLINE

SPLINE
SPL {X  -105.077, Y  +256.854, Z    +0.000, E1   +55.187, E3 +98298.924}
SPL {X  -133.208, Y  +288.886, Z    +0.000, E1   +52.003, E3 +98332.025}
SPL {X  -149.825, Y  +321.381, Z    +0.000, E1   +42.580, E3 +98345.178}
SPL {X  -157.376, Y  +348.695, Z    +0.000, E1   +27.651, E3 +98350.263}
SPL {X  -159.486, Y  +364.808, Z    +0.000, E1   +14.693, E3 +98351.767}
SPL {X  -159.964, Y  +374.630, Z    +0.000, E1    +5.249, E3 +98352.172}
SPL {X  -159.990, Y  +379.484, Z    +0.000, E1    +0.034, E3 +98352.228}
SPL {X  -159.990, Y  +381.639, Z    +0.000, E1    -4.454, E3 +98352.249}
SPL {X  -159.990, Y  +385.871, Z    +0.000, E1   -15.161, E3 +98352.365}
SPL {X  -159.990, Y  +391.065, Z    +0.000, E1   -28.187, E3 +98352.653}
SPL {X  -159.990, Y  +399.326, Z    +0.000, E1   -44.934, E3 +98353.437}
SPL {X  -159.990, Y  +408.817, Z    +0.000, E1   -56.572, E3 +98354.809}
SPL {X  -159.990, Y  +426.617, Z    +0.000, E1   -66.230, E3 +98358.665}
SPL {X  -159.990, Y  +499.521, Z    +0.000, E1   -73.662, E3 +98381.991}
SPL {X  -159.629, Y  +687.249, Z    +0.000, E1   -74.539, E3 +98469.875}
SPL {X  -157.983, Y  +701.765, Z    +0.000, E1   -74.384, E3 +98480.108}
SPL {X  -155.520, Y  +714.054, Z    +0.000, E1   -74.151, E3 +98489.862}
SPL {X  -152.569, Y  +724.660, Z    +0.000, E1   -73.857, E3 +98499.096}
SPL {X  -149.625, Y  +733.149, Z    +0.000, E1   -73.553, E3 +98507.032}
SPL {X  -146.617, Y  +740.532, Z    +0.000, E1   -73.233, E3 +98514.308}
SPL {X  -143.394, Y  +747.457, Z    +0.000, E1   -72.883, E3 +98521.405}
SPL {X  -140.332, Y  +753.336, Z    +0.000, E1   -72.527, E3 +98527.680}
SPL {X  -137.187, Y  +758.820, Z    +0.000, E1   -72.156, E3 +98533.683}
SPL {X  -134.014, Y  +763.891, Z    +0.000, E1   -71.759, E3 +98539.368}
SPL {X  -130.657, Y  +768.834, Z    +0.000, E1   -71.330, E3 +98544.984}
SPL {X  -126.020, Y  +775.068, Z    +0.000, E1   -70.718, E3 +98552.111}
SPL {X  -121.287, Y  +780.838, Z    +0.000, E1   -70.013, E3 +98558.685}
SPL {X   -75.772, Y  +817.409, Z    +0.000, E1   -56.226, E3 +98686.037}
ENDSPLINE

SPLINE
SPL {X  -124.054, Y  +777.532, Z    +0.000, E1   -54.436, E3 +98869.265}
SPL {X  -149.719, Y  +732.901, Z    +0.000, E1   -43.150, E3 +98890.080}
SPL {X  -158.004, Y  +701.630, Z    +0.000, E1   -25.366, E3 +98895.544}
SPL {X  -159.639, Y  +687.095, Z    +0.000, E1   -12.931, E3 +98896.702}
SPL {X  -159.981, Y  +678.202, Z    +0.000, E1    -4.129, E3 +98896.996}
SPL {X  -159.990, Y  +674.500, Z    +0.000, E1    +0.000, E3 +98897.034}
SPL {X  -159.990, Y  +672.677, Z    +0.000, E1    +3.879, E3 +98897.049}
SPL {X  -159.990, Y  +669.117, Z    +0.000, E1   +12.900, E3 +98897.132}
SPL {X  -159.990, Y  +665.253, Z    +0.000, E1   +22.908, E3 +98897.306}
SPL {X  -159.990, Y  +658.335, Z    +0.000, E1   +38.839, E3 +98897.850}
SPL {X  -159.990, Y  +645.786, Z    +0.000, E1   +56.338, E3 +98899.565}
SPL {X  -159.990, Y  +623.264, Z    +0.000, E1   +67.753, E3 +98904.490}
SPL {X  -159.990, Y  +547.268, Z    +0.000, E1   +73.735, E3 +98930.178}
SPL {X  -159.626, Y  +366.721, Z    +0.000, E1   +74.756, E3 +99012.444}
SPL {X  -157.975, Y  +352.185, Z    +0.000, E1   +74.622, E3 +99022.510}
SPL {X  -154.546, Y  +336.120, Z    +0.000, E1   +74.400, E3 +99034.168}
SPL {X  -141.909, Y  +303.617, Z    +0.000, E1   +76.515, E3 +99029.135}
ENDSPLINE

SPLINE
SPL {X  -142.567, Y  +304.895, Z    +0.000, E1   +75.566, E3 +99037.950}
ENDSPLINE

SPLINE
SPL {X  -141.999, Y  +303.790, Z    +0.000, E1   +74.633, E3 +99047.201}
SPL {X  -141.780, Y  +303.371, Z    +0.000, E1   +73.549, E3 +99056.775}
SPL {X  -140.619, Y  +301.190, Z    +0.000, E1   +72.741, E3 +99064.622}
SPL {X  -137.438, Y  +295.601, Z    +0.000, E1   +72.365, E3 +99070.710}
SPL {X  -134.156, Y  +290.328, Z    +0.000, E1   +71.962, E3 +99076.581}
SPL {X  -130.677, Y  +285.194, Z    +0.000, E1   +71.519, E3 +99082.386}
SPL {X  -127.147, Y  +280.390, Z    +0.000, E1   +71.042, E3 +99087.870}
SPL {X  -123.431, Y  +275.709, Z    +0.000, E1   +70.518, E3 +99093.193}
SPL {X  -120.392, Y  +272.131, Z    +0.000, E1   +70.053, E3 +99097.214}
SPL {X   -79.311, Y  +238.552, Z    +0.000, E1   +58.563, E3 +99192.453}
ENDSPLINE

SPLINE
SPL {X  -105.077, Y  +256.854, Z    +0.000, E1   +55.187, E3 +99380.005}
SPL {X  -133.208, Y  +288.886, Z    +0.000, E1   +52.003, E3 +99413.106}
SPL {X  -149.825, Y  +321.381, Z    +0.000, E1   +42.580, E3 +99426.260}
SPL {X  -156.491, Y  +344.222, Z    +0.000, E1   +30.612, E3 +99430.766}
SPL {X  -159.275, Y  +362.387, Z    +0.000, E1   +16.907, E3 +99432.680}
SPL {X  -159.964, Y  +374.630, Z    +0.000, E1    +5.249, E3 +99433.253}
SPL {X  -159.990, Y  +379.735, Z    +0.000, E1    -0.236, E3 +99433.310}
SPL {X  -159.990, Y  +382.878, Z    +0.000, E1    -7.664, E3 +99433.349}
SPL {X  -159.990, Y  +387.459, Z    +0.000, E1   -18.927, E3 +99433.526}
SPL {X  -159.990, Y  +395.361, Z    +0.000, E1   -37.740, E3 +99434.091}
SPL {X  -159.990, Y  +406.369, Z    +0.000, E1   -54.148, E3 +99435.496}
SPL {X  -159.990, Y  +426.617, Z    +0.000, E1   -66.230, E3 +99439.746}
SPL {X  -159.990, Y  +499.521, Z    +0.000, E1   -73.662, E3 +99463.072}
SPL {X  -159.629, Y  +687.249, Z    +0.000, E1   -74.539, E3 +99550.957}
SPL {X  -157.983, Y  +701.765, Z    +0.000, E1   -74.384, E3 +99561.189}
SPL {X  -155.520, Y  +714.054, Z    +0.000, E1   -74.151, E3 +99570.943}
SPL {X  -152.569, Y  +724.660, Z    +0.000, E1   -73.857, E3 +99580.177}
SPL {X  -149.625, Y  +733.149, Z    +0.000, E1   -73.553, E3 +99588.113}
SPL {X  -146.617, Y  +740.532, Z    +0.000, E1   -73.233, E3 +99595.389}
SPL {X  -143.394, Y  +747.457, Z    +0.000, E1   -72.883, E3 +99602.486}
SPL {X  -140.332, Y  +753.336, Z    +0.000, E1   -72.527, E3 +99608.761}
SPL {X  -137.187, Y  +758.820, Z    +0.000, E1   -72.156, E3 +99614.764}
SPL {X  -134.014, Y  +763.891, Z    +0.000, E1   -71.759, E3 +99620.450}
SPL {X  -130.657, Y  +768.834, Z    +0.000, E1   -71.330, E3 +99626.065}
SPL {X  -126.937, Y  +773.885, Z    +0.000, E1   -70.823, E3 +99631.867}
SPL {X  -122.983, Y  +778.833, Z    +0.000, E1   -70.262, E3 +99637.511}
SPL {X  -120.205, Y  +782.082, Z    +0.000, E1   -69.822, E3 +99641.180}
SPL {X   -75.772, Y  +817.409, Z    +0.000, E1   -56.226, E3 +99767.119}
ENDSPLINE

SPLINE
SPL {X  -124.054, Y  +777.532, Z    +0.000, E1   -54.436, E3 +99950.346}
SPL {X  -145.922, Y  +742.101, Z    +0.000, E1   -46.535, E3 +99968.616}
SPL {X  -155.216, Y  +715.293, Z    +0.000, E1   -34.460, E3 +99974.808}
SPL {X  -159.282, Y  +691.530, Z    +0.000, E1   -17.100, E3 +99977.503}
SPL {X  -159.981, Y  +678.202, Z    +0.000, E1    -4.129, E3 +99978.077}
SPL {X  -159.990, Y  +674.500, Z    +0.000, E1    +0.000, E3 +99978.115}
SPL {X  -159.990, Y  +672.677, Z    +0.000, E1    +3.879, E3 +99978.130}
SPL {X  -159.990, Y  +669.117, Z    +0.000, E1   +12.900, E3 +99978.213}
SPL {X  -159.990, Y  +665.253, Z    +0.000, E1   +22.908, E3 +99978.387}
SPL {X  -159.990, Y  +658.335, Z    +0.000, E1   +38.839, E3 +99978.931}
SPL {X  -159.990, Y  +645.786, Z    +0.000, E1   +56.338, E3 +99980.646}
SPL {X  -159.990, Y  +623.264, Z    +0.000, E1   +67.753, E3 +99985.571}
SPL {X  -159.990, Y  +547.268, Z    +0.000, E1   +73.735, E3 +100011.260}
SPL {X  -159.091, Y  +360.560, Z    +0.000, E1   +74.726, E3 +100097.586}
SPL {X  -156.418, Y  +343.879, Z    +0.000, E1   +74.473, E3 +100110.011}
SPL {X  -153.414, Y  +332.103, Z    +0.000, E1   +74.378, E3 +100117.686}
SPL {X  -141.909, Y  +303.617, Z    +0.000, E1   +76.515, E3 +100110.216}
ENDSPLINE

SPLINE
SPL {X  -142.567, Y  +304.895, Z    +0.000, E1   +75.566, E3 +100119.031}
ENDSPLINE

SPLINE
SPL {X  -141.999, Y  +303.790, Z    +0.000, E1   +74.633, E3 +100128.282}
SPL {X  -141.780, Y  +303.371, Z    +0.000, E1   +73.549, E3 +100137.856}
SPL {X  -140.619, Y  +301.190, Z    +0.000, E1   +72.741, E3 +100145.703}
SPL {X  -137.438, Y  +295.601, Z    +0.000, E1   +72.365, E3 +100151.791}
SPL {X  -134.156, Y  +290.328, Z    +0.000, E1   +71.962, E3 +100157.662}
SPL {X  -130.677, Y  +285.194, Z    +0.000, E1   +71.519, E3 +100163.467}
SPL {X  -126.239, Y  +279.212, Z    +0.000, E1   +70.937, E3 +100170.268}
SPL {X  -121.335, Y  +273.218, Z    +0.000, E1   +70.225, E3 +100177.056}
SPL {X   -79.311, Y  +238.552, Z    +0.000, E1   +58.563, E3 +100273.534}
ENDSPLINE

SPLINE
SPL {X  -105.077, Y  +256.854, Z    +0.000, E1   +55.187, E3 +100461.086}
SPL {X  -133.208, Y  +288.886, Z    +0.000, E1   +52.003, E3 +100494.187}
SPL {X  -149.825, Y  +321.381, Z    +0.000, E1   +42.580, E3 +100507.341}
SPL {X  -156.491, Y  +344.222, Z    +0.000, E1   +30.612, E3 +100511.847}
SPL {X  -159.275, Y  +362.387, Z    +0.000, E1   +16.907, E3 +100513.761}
SPL {X  -159.964, Y  +374.630, Z    +0.000, E1    +5.249, E3 +100514.334}
SPL {X  -159.990, Y  +379.484, Z    +0.000, E1    +0.034, E3 +100514.390}
SPL {X  -159.990, Y  +381.639, Z    +0.000, E1    -4.454, E3 +100514.412}
SPL {X  -159.990, Y  +385.871, Z    +0.000, E1   -15.161, E3 +100514.528}
SPL {X  -159.990, Y  +391.065, Z    +0.000, E1   -28.187, E3 +100514.815}
SPL {X  -159.990, Y  +397.286, Z    +0.000, E1   -41.591, E3 +100515.358}
SPL {X  -159.990, Y  +406.369, Z    +0.000, E1   -54.148, E3 +100516.577}
SPL {X  -159.990, Y  +426.617, Z    +0.000, E1   -66.230, E3 +100520.827}
SPL {X  -159.990, Y  +499.521, Z    +0.000, E1   -73.662, E3 +100544.153}
SPL {X  -159.629, Y  +687.249, Z    +0.000, E1   -74.539, E3 +100632.038}
SPL {X  -157.983, Y  +701.765, Z    +0.000, E1   -74.384, E3 +100642.270}
SPL {X  -155.520, Y  +714.054, Z    +0.000, E1   -74.151, E3 +100652.024}
SPL {X  -152.569, Y  +724.660, Z    +0.000, E1   -73.857, E3 +100661.258}
SPL {X  -149.625, Y  +733.149, Z    +0.000, E1   -73.553, E3 +100669.194}
SPL {X  -146.617, Y  +740.532, Z    +0.000, E1   -73.233, E3 +100676.470}
SPL {X  -143.394, Y  +747.457, Z    +0.000, E1   -72.883, E3 +100683.567}
SPL {X  -140.332, Y  +753.336, Z    +0.000, E1   -72.527, E3 +100689.842}
SPL {X  -137.187, Y  +758.820, Z    +0.000, E1   -72.156, E3 +100695.845}
SPL {X  -134.014, Y  +763.891, Z    +0.000, E1   -71.759, E3 +100701.531}
SPL {X  -130.657, Y  +768.834, Z    +0.000, E1   -71.330, E3 +100707.146}
SPL {X  -126.020, Y  +775.068, Z    +0.000, E1   -70.718, E3 +100714.274}
SPL {X  -121.287, Y  +780.838, Z    +0.000, E1   -70.013, E3 +100720.847}
SPL {X   -75.772, Y  +817.409, Z    +0.000, E1   -56.226, E3 +100848.200}
ENDSPLINE

SPLINE
SPL {X  -124.054, Y  +777.532, Z    +0.000, E1   -54.436, E3 +101031.427}
SPL {X  -149.719, Y  +732.901, Z    +0.000, E1   -43.150, E3 +101052.242}
SPL {X  -158.004, Y  +701.630, Z    +0.000, E1   -25.366, E3 +101057.706}
SPL {X  -159.639, Y  +687.095, Z    +0.000, E1   -12.931, E3 +101058.865}
SPL {X  -159.981, Y  +678.202, Z    +0.000, E1    -4.129, E3 +101059.158}
SPL {X  -159.990, Y  +674.500, Z    +0.000, E1    +0.000, E3 +101059.196}
SPL {X  -159.990, Y  +672.677, Z    +0.000, E1    +3.879, E3 +101059.211}
SPL {X  -159.990, Y  +669.117, Z    +0.000, E1   +12.900, E3 +101059.294}
SPL {X  -159.990, Y  +665.253, Z    +0.000, E1   +22.908, E3 +101059.468}
SPL {X  -159.990, Y  +658.335, Z    +0.000, E1   +38.839, E3 +101060.012}
SPL {X  -159.990, Y  +645.786, Z    +0.000, E1   +56.338, E3 +101061.727}
SPL {X  -159.990, Y  +623.264, Z    +0.000, E1   +67.753, E3 +101066.652}
SPL {X  -159.990, Y  +547.268, Z    +0.000, E1   +73.735, E3 +101092.341}
SPL {X  -159.091, Y  +360.560, Z    +0.000, E1   +74.726, E3 +101178.667}
SPL {X  -156.418, Y  +343.879, Z    +0.000, E1   +74.473, E3 +101191.092}
SPL {X  -153.414, Y  +332.103, Z    +0.000, E1   +74.378, E3 +101198.767}
SPL {X  -141.909, Y  +303.617, Z    +0.000, E1   +76.515, E3 +101191.297}
ENDSPLINE

SPLINE
SPL {X  -142.567, Y  +304.895, Z    +0.000, E1   +75.566, E3 +101200.112}
ENDSPLINE

SPLINE
SPL {X  -141.999, Y  +303.790, Z    +0.000, E1   +74.633, E3 +101209.363}
SPL {X  -141.780, Y  +303.371, Z    +0.000, E1   +73.549, E3 +101218.937}
SPL {X  -140.619, Y  +301.190, Z    +0.000, E1   +72.741, E3 +101226.784}
SPL {X  -137.438, Y  +295.601, Z    +0.000, E1   +72.365, E3 +101232.872}
SPL {X  -134.156, Y  +290.328, Z    +0.000, E1   +71.962, E3 +101238.743}
SPL {X  -130.677, Y  +285.194, Z    +0.000, E1   +71.519, E3 +101244.548}
SPL {X  -126.239, Y  +279.212, Z    +0.000, E1   +70.937, E3 +101251.349}
SPL {X  -121.335, Y  +273.218, Z    +0.000, E1   +70.225, E3 +101258.137}
SPL {X   -79.311, Y  +238.552, Z    +0.000, E1   +58.563, E3 +101354.615}
ENDSPLINE

SPLINE
SPL {X  -105.077, Y  +256.854, Z    +0.000, E1   +55.187, E3 +101542.167}
SPL {X  -133.208, Y  +288.886, Z    +0.000, E1   +52.003, E3 +101575.268}
SPL {X  -149.825, Y  +321.381, Z    +0.000, E1   +42.580, E3 +101588.422}
SPL {X  -156.491, Y  +344.222, Z    +0.000, E1   +30.612, E3 +101592.928}
SPL {X  -159.275, Y  +362.387, Z    +0.000, E1   +16.907, E3 +101594.842}
SPL {X  -159.964, Y  +374.630, Z    +0.000, E1    +5.249, E3 +101595.415}
SPL {X  -159.990, Y  +379.484, Z    +0.000, E1    +0.034, E3 +101595.471}
SPL {X  -159.990, Y  +381.639, Z    +0.000, E1    -4.454, E3 +101595.493}
SPL {X  -159.990, Y  +385.871, Z    +0.000, E1   -15.161, E3 +101595.609}
SPL {X  -159.990, Y  +391.065, Z    +0.000, E1   -28.187, E3 +101595.897}
SPL {X  -159.990, Y  +397.286, Z    +0.000, E1   -41.591, E3 +101596.439}
SPL {X  -159.990, Y  +406.369, Z    +0.000, E1   -54.148, E3 +101597.658}
SPL {X  -159.990, Y  +426.617, Z    +0.000, E1   -66.230, E3 +101601.908}
SPL {X  -159.990, Y  +499.521, Z    +0.000, E1   -73.662, E3 +101625.234}
SPL {X  -159.629, Y  +687.249, Z    +0.000, E1   -74.539, E3 +101713.119}
SPL {X  -157.983, Y  +701.765, Z    +0.000, E1   -74.384, E3 +101723.351}
SPL {X  -155.520, Y  +714.054, Z    +0.000, E1   -74.151, E3 +101733.105}
SPL {X  -152.569, Y  +724.660, Z    +0.000, E1   -73.857, E3 +101742.340}
SPL {X  -149.625, Y  +733.149, Z    +0.000, E1   -73.553, E3 +101750.275}
SPL {X  -146.617, Y  +740.532, Z    +0.000, E1   -73.233, E3 +101757.551}
SPL {X  -143.394, Y  +747.457, Z    +0.000, E1   -72.883, E3 +101764.648}
SPL {X  -140.332, Y  +753.336, Z    +0.000, E1   -72.527, E3 +101770.923}
SPL {X  -137.187, Y  +758.820, Z    +0.000, E1   -72.156, E3 +101776.926}
SPL {X  -134.014, Y  +763.891, Z    +0.000, E1   -71.759, E3 +101782.612}
SPL {X  -130.657, Y  +768.834, Z    +0.000, E1   -71.330, E3 +101788.227}
SPL {X  -126.937, Y  +773.885, Z    +0.000, E1   -70.823, E3 +101794.029}
SPL {X  -122.983, Y  +778.833, Z    +0.000, E1   -70.262, E3 +101799.673}
SPL {X  -120.205, Y  +782.082, Z    +0.000, E1   -69.822, E3 +101803.342}
SPL {X   -77.717, Y  +816.346, Z    +0.000, E1   -57.422, E3 +101911.193}
SPL {X   -74.440, Y  +818.117, Z    +0.000, E1   -54.647, E3 +101964.432}
ENDSPLINE

SPLINE
SPL {X  -124.054, Y  +777.532, Z    +0.000, E1   -54.436, E3 +102112.508}
SPL {X  -149.719, Y  +732.901, Z    +0.000, E1   -43.150, E3 +102133.323}
SPL {X  -158.004, Y  +701.630, Z    +0.000, E1   -25.366, E3 +102138.788}
SPL {X  -159.838, Y  +683.473, Z    +0.000, E1    -9.532, E3 +102140.094}
SPL {X  -159.990, Y  +674.579, Z    +0.000, E1    -0.168, E3 +102140.277}
SPL {X  -159.990, Y  +672.677, Z    +0.000, E1    +3.879, E3 +102140.292}
SPL {X  -159.990, Y  +669.117, Z    +0.000, E1   +12.900, E3 +102140.375}
SPL {X  -159.990, Y  +665.253, Z    +0.000, E1   +22.908, E3 +102140.549}
SPL {X  -159.990, Y  +658.335, Z    +0.000, E1   +38.839, E3 +102141.094}
SPL {X  -159.990, Y  +645.786, Z    +0.000, E1   +56.338, E3 +102142.808}
SPL {X  -159.990, Y  +623.264, Z    +0.000, E1   +67.753, E3 +102147.734}
SPL {X  -159.990, Y  +547.268, Z    +0.000, E1   +73.735, E3 +102173.422}
SPL {X  -159.091, Y  +360.560, Z    +0.000, E1   +74.726, E3 +102259.748}
SPL {X  -156.418, Y  +343.879, Z    +0.000, E1   +74.473, E3 +102272.173}
SPL {X  -153.414, Y  +332.103, Z    +0.000, E1   +74.378, E3 +102279.848}
SPL {X  -141.909, Y  +303.617, Z    +0.000, E1   +76.515, E3 +102272.378}
ENDSPLINE

SPLINE
SPL {X  -142.567, Y  +304.895, Z    +0.000, E1   +75.566, E3 +102281.193}
ENDSPLINE

SPLINE
SPL {X  -141.999, Y  +303.790, Z    +0.000, E1   +74.633, E3 +102290.445}
SPL {X  -141.780, Y  +303.371, Z    +0.000, E1   +73.549, E3 +102300.018}
SPL {X  -140.619, Y  +301.190, Z    +0.000, E1   +72.741, E3 +102307.865}
SPL {X  -137.438, Y  +295.601, Z    +0.000, E1   +72.365, E3 +102313.953}
SPL {X  -134.156, Y  +290.328, Z    +0.000, E1   +71.962, E3 +102319.824}
SPL {X  -130.677, Y  +285.194, Z    +0.000, E1   +71.519, E3 +102325.629}
SPL {X  -127.147, Y  +280.390, Z    +0.000, E1   +71.042, E3 +102331.113}
SPL {X  -123.431, Y  +275.709, Z    +0.000, E1   +70.518, E3 +102336.436}
SPL {X  -120.392, Y  +272.131, Z    +0.000, E1   +70.053, E3 +102340.457}
SPL {X   -79.311, Y  +238.552, Z    +0.000, E1   +58.563, E3 +102435.696}
ENDSPLINE

SPLINE
SPL {X  -105.077, Y  +256.854, Z    +0.000, E1   +55.187, E3 +102623.248}
SPL {X  -133.208, Y  +288.886, Z    +0.000, E1   +52.003, E3 +102656.349}
SPL {X  -149.825, Y  +321.381, Z    +0.000, E1   +42.580, E3 +102669.503}
SPL {X  -157.376, Y  +348.695, Z    +0.000, E1   +27.651, E3 +102674.588}
SPL {X  -159.486, Y  +364.808, Z    +0.000, E1   +14.693, E3 +102676.091}
SPL {X  -159.964, Y  +374.630, Z    +0.000, E1    +5.249, E3 +102676.496}
SPL {X  -159.990, Y  +379.484, Z    +0.000, E1    +0.034, E3 +102676.552}
SPL {X  -159.990, Y  +381.639, Z    +0.000, E1    -4.454, E3 +102676.574}
SPL {X  -159.990, Y  +387.459, Z    +0.000, E1   -18.927, E3 +102676.770}
SPL {X  -159.990, Y  +393.138, Z    +0.000, E1   -33.246, E3 +102677.119}
SPL {X  -159.990, Y  +399.326, Z    +0.000, E1   -44.934, E3 +102677.761}
SPL {X  -159.990, Y  +408.817, Z    +0.000, E1   -56.572, E3 +102679.134}
SPL {X  -159.990, Y  +426.617, Z    +0.000, E1   -66.230, E3 +102682.989}
SPL {X  -159.990, Y  +499.521, Z    +0.000, E1   -73.662, E3 +102706.316}
SPL {X  -159.629, Y  +687.249, Z    +0.000, E1   -74.539, E3 +102794.200}
SPL {X  -157.983, Y  +701.765, Z    +0.000, E1   -74.384, E3 +102804.432}
SPL {X  -155.520, Y  +714.054, Z    +0.000, E1   -74.151, E3 +102814.186}
SPL {X  -152.569, Y  +724.660, Z    +0.000, E1   -73.857, E3 +102823.421}
SPL {X  -149.625, Y  +733.149, Z    +0.000, E1   -73.553, E3 +102831.356}
SPL {X  -146.617, Y  +740.532, Z    +0.000, E1   -73.233, E3 +102838.632}
SPL {X  -143.394, Y  +747.457, Z    +0.000, E1   -72.883, E3 +102845.729}
SPL {X  -140.332, Y  +753.336, Z    +0.000, E1   -72.527, E3 +102852.004}
SPL {X  -137.187, Y  +758.820, Z    +0.000, E1   -72.156, E3 +102858.007}
SPL {X  -134.014, Y  +763.891, Z    +0.000, E1   -71.759, E3 +102863.693}
SPL {X  -130.657, Y  +768.834, Z    +0.000, E1   -71.330, E3 +102869.308}
SPL {X  -126.937, Y  +773.885, Z    +0.000, E1   -70.823, E3 +102875.110}
SPL {X  -122.983, Y  +778.833, Z    +0.000, E1   -70.262, E3 +102880.755}
SPL {X  -120.205, Y  +782.082, Z    +0.000, E1   -69.822, E3 +102884.423}
SPL {X   -75.772, Y  +817.409, Z    +0.000, E1   -56.226, E3 +103010.362}
ENDSPLINE

SPLINE
SPL {X  -124.054, Y  +777.532, Z    +0.000, E1   -54.436, E3 +103193.590}
SPL {X  -145.922, Y  +742.101, Z    +0.000, E1   -46.535, E3 +103211.859}
SPL {X  -155.216, Y  +715.293, Z    +0.000, E1   -34.460, E3 +103218.052}
SPL {X  -159.282, Y  +691.530, Z    +0.000, E1   -17.100, E3 +103220.747}
SPL {X  -159.981, Y  +678.202, Z    +0.000, E1    -4.129, E3 +103221.321}
SPL {X  -159.990, Y  +674.500, Z    +0.000, E1    +0.000, E3 +103221.358}
SPL {X  -159.990, Y  +672.677, Z    +0.000, E1    +3.879, E3 +103221.374}
SPL {X  -159.990, Y  +669.117, Z    +0.000, E1   +12.900, E3 +103221.456}
SPL {X  -159.990, Y  +665.253, Z    +0.000, E1   +22.908, E3 +103221.630}
SPL {X  -159.990, Y  +658.335, Z    +0.000, E1   +38.839, E3 +103222.175}
SPL {X  -159.990, Y  +645.786, Z    +0.000, E1   +56.338, E3 +103223.889}
SPL {X  -159.990, Y  +623.264, Z    +0.000, E1   +67.753, E3 +103228.815}
SPL {X  -159.990, Y  +547.268, Z    +0.000, E1   +73.735, E3 +103254.503}
SPL {X  -159.091, Y  +360.560, Z    +0.000, E1   +74.726, E3 +103340.829}
SPL {X  -156.418, Y  +343.879, Z    +0.000, E1   +74.473, E3 +103353.255}
SPL {X  -153.414, Y  +332.103, Z    +0.000, E1   +74.378, E3 +103360.929}
SPL {X  -141.909, Y  +303.617, Z    +0.000, E1   +76.515, E3 +103353.459}
ENDSPLINE

SPLINE
SPL {X  -142.567, Y  +304.895, Z    +0.000, E1   +75.566, E3 +103362.274}
ENDSPLINE

SPLINE
SPL {X  -141.999, Y  +303.790, Z    +0.000, E1   +74.633, E3 +103371.526}
SPL {X  -141.780, Y  +303.371, Z    +0.000, E1   +73.549, E3 +103381.099}
SPL {X  -140.619, Y  +301.190, Z    +0.000, E1   +72.741, E3 +103388.946}
SPL {X  -137.438, Y  +295.601, Z    +0.000, E1   +72.365, E3 +103395.034}
SPL {X  -134.156, Y  +290.328, Z    +0.000, E1   +71.962, E3 +103400.905}
SPL {X  -130.677, Y  +285.194, Z    +0.000, E1   +71.519, E3 +103406.710}
SPL {X  -126.239, Y  +279.212, Z    +0.000, E1   +70.937, E3 +103413.511}
SPL {X  -121.335, Y  +273.218, Z    +0.000, E1   +70.225, E3 +103420.299}
SPL {X   -79.311, Y  +238.552, Z    +0.000, E1   +58.563, E3 +103516.777}
ENDSPLINE

SPLINE
SPL {X  -105.077, Y  +256.854, Z    +0.000, E1   +55.187, E3 +103704.329}
SPL {X  -133.208, Y  +288.886, Z    +0.000, E1   +52.003, E3 +103737.430}
SPL {X  -149.825, Y  +321.381, Z    +0.000, E1   +42.580, E3 +103750.584}
SPL {X  -156.491, Y  +344.222, Z    +0.000, E1   +30.612, E3 +103755.090}
SPL {X  -159.275, Y  +362.387, Z    +0.000, E1   +16.907, E3 +103757.004}
SPL {X  -159.964, Y  +374.630, Z    +0.000, E1    +5.249, E3 +103757.577}
SPL {X  -159.990, Y  +379.484, Z    +0.000, E1    +0.034, E3 +103757.633}
SPL {X  -159.990, Y  +381.639, Z    +0.000, E1    -4.454, E3 +103757.655}
SPL {X  -159.990, Y  +385.871, Z    +0.000, E1   -15.161, E3 +103757.771}
SPL {X  -159.990, Y  +391.065, Z    +0.000, E1   -28.187, E3 +103758.059}
SPL {X  -159.990, Y  +397.286, Z    +0.000, E1   -41.591, E3 +103758.601}
SPL {X  -159.990, Y  +406.369, Z    +0.000, E1   -54.148, E3 +103759.820}
SPL {X  -159.990, Y  +426.617, Z    +0.000, E1   -66.230, E3 +103764.070}
SPL {X  -159.990, Y  +499.521, Z    +0.000, E1   -73.662, E3 +103787.397}
SPL {X  -159.629, Y  +687.249, Z    +0.000, E1   -74.539, E3 +103875.281}
SPL {X  -157.983, Y  +701.765, Z    +0.000, E1   -74.384, E3 +103885.513}
SPL {X  -155.520, Y  +714.054, Z    +0.000, E1   -74.151, E3 +103895.267}
SPL {X  -152.569, Y  +724.660, Z    +0.000, E1   -73.857, E3 +103904.502}
SPL {X  -149.625, Y  +733.149, Z    +0.000, E1   -73.553, E3 +103912.437}
SPL {X  -146.617, Y  +740.532, Z    +0.000, E1   -73.233, E3 +103919.713}
SPL {X  -143.394, Y  +747.457, Z    +0.000, E1   -72.883, E3 +103926.810}
SPL {X  -140.332, Y  +753.336, Z    +0.000, E1   -72.527, E3 +103933.085}
SPL {X  -137.187, Y  +758.820, Z    +0.000, E1   -72.156, E3 +103939.088}
SPL {X  -134.014, Y  +763.891, Z    +0.000, E1   -71.759, E3 +103944.774}
SPL {X  -130.657, Y  +768.834, Z    +0.000, E1   -71.330, E3 +103950.389}
SPL {X  -126.020, Y  +775.068, Z    +0.000, E1   -70.718, E3 +103957.517}
SPL {X  -121.287, Y  +780.838, Z    +0.000, E1   -70.013, E3 +103964.090}
SPL {X   -75.772, Y  +817.409, Z    +0.000, E1   -56.226, E3 +104091.443}
ENDSPLINE

SPLINE
SPL {X  -124.054, Y  +777.532, Z    +0.000, E1   -54.436, E3 +104274.671}
SPL {X  -149.719, Y  +732.901, Z    +0.000, E1   -43.150, E3 +104295.485}
SPL {X  -158.004, Y  +701.630, Z    +0.000, E1   -25.366, E3 +104300.950}
SPL {X  -159.639, Y  +687.095, Z    +0.000, E1   -12.931, E3 +104302.108}
SPL {X  -159.981, Y  +678.202, Z    +0.000, E1    -4.129, E3 +104302.402}
SPL {X  -159.990, Y  +674.500, Z    +0.000, E1    +0.000, E3 +104302.439}
SPL {X  -159.990, Y  +672.677, Z    +0.000, E1    +3.879, E3 +104302.455}
SPL {X  -159.990, Y  +669.117, Z    +0.000, E1   +12.900, E3 +104302.537}
SPL {X  -159.990, Y  +665.253, Z    +0.000, E1   +22.908, E3 +104302.711}
SPL {X  -159.990, Y  +658.335, Z    +0.000, E1   +38.839, E3 +104303.256}
SPL {X  -159.990, Y  +645.786, Z    +0.000, E1   +56.338, E3 +104304.970}
SPL {X  -159.990, Y  +623.264, Z    +0.000, E1   +67.753, E3 +104309.896}
SPL {X  -159.990, Y  +547.268, Z    +0.000, E1   +73.735, E3 +104335.584}
SPL {X  -159.091, Y  +360.560, Z    +0.000, E1   +74.726, E3 +104421.910}
SPL {X  -156.418, Y  +343.879, Z    +0.000, E1   +74.473, E3 +104434.336}
SPL {X  -153.414, Y  +332.103, Z    +0.000, E1   +74.378, E3 +104442.010}
SPL {X  -141.909, Y  +303.617, Z    +0.000, E1   +76.515, E3 +104434.540}
ENDSPLINE

SPLINE
SPL {X  -142.567, Y  +304.895, Z    +0.000, E1   +75.566, E3 +104443.355}
ENDSPLINE

SPLINE
SPL {X  -141.999, Y  +303.790, Z    +0.000, E1   +74.633, E3 +104452.607}
SPL {X  -141.780, Y  +303.371, Z    +0.000, E1   +73.549, E3 +104462.180}
SPL {X  -140.619, Y  +301.190, Z    +0.000, E1   +72.741, E3 +104470.027}
SPL {X  -137.438, Y  +295.601, Z    +0.000, E1   +72.365, E3 +104476.115}
SPL {X  -134.156, Y  +290.328, Z    +0.000, E1   +71.962, E3 +104481.986}
SPL {X  -130.677, Y  +285.194, Z    +0.000, E1   +71.519, E3 +104487.791}
SPL {X  -126.239, Y  +279.212, Z    +0.000, E1   +70.937, E3 +104494.592}
SPL {X  -121.335, Y  +273.218, Z    +0.000, E1   +70.225, E3 +104501.381}
SPL {X   -79.311, Y  +238.552, Z    +0.000, E1   +58.563, E3 +104597.858}
ENDSPLINE

SPLINE
SPL {X  -105.077, Y  +256.854, Z    +0.000, E1   +55.187, E3 +104785.410}
SPL {X  -133.208, Y  +288.886, Z    +0.000, E1   +52.003, E3 +104818.511}
SPL {X  -149.825, Y  +321.381, Z    +0.000, E1   +42.580, E3 +104831.665}
SPL {X  -156.491, Y  +344.222, Z    +0.000, E1   +30.612, E3 +104836.171}
SPL {X  -159.275, Y  +362.387, Z    +0.000, E1   +16.907, E3 +104838.085}
SPL {X  -159.964, Y  +374.630, Z    +0.000, E1    +5.249, E3 +104838.658}
SPL {X  -159.990, Y  +379.484, Z    +0.000, E1    +0.034, E3 +104838.714}
SPL {X  -159.990, Y  +381.639, Z    +0.000, E1    -4.454, E3 +104838.736}
SPL {X  -159.990, Y  +385.871, Z    +0.000, E1   -15.161, E3 +104838.852}
SPL {X  -159.990, Y  +391.065, Z    +0.000, E1   -28.187, E3 +104839.140}
SPL {X  -159.990, Y  +397.286, Z    +0.000, E1   -41.591, E3 +104839.682}
SPL {X  -159.990, Y  +406.369, Z    +0.000, E1   -54.148, E3 +104840.901}
SPL {X  -159.990, Y  +426.617, Z    +0.000, E1   -66.230, E3 +104845.151}
SPL {X  -159.990, Y  +499.521, Z    +0.000, E1   -73.662, E3 +104868.478}
SPL {X  -159.629, Y  +687.249, Z    +0.000, E1   -74.539, E3 +104956.362}
SPL {X  -157.983, Y  +701.765, Z    +0.000, E1   -74.384, E3 +104966.594}
SPL {X  -155.520, Y  +714.054, Z    +0.000, E1   -74.151, E3 +104976.348}
SPL {X  -152.569, Y  +724.660, Z    +0.000, E1   -73.857, E3 +104985.583}
SPL {X  -149.625, Y  +733.149, Z    +0.000, E1   -73.553, E3 +104993.518}
SPL {X  -146.617, Y  +740.532, Z    +0.000, E1   -73.233, E3 +105000.794}
SPL {X  -143.394, Y  +747.457, Z    +0.000, E1   -72.883, E3 +105007.891}
SPL {X  -140.332, Y  +753.336, Z    +0.000, E1   -72.527, E3 +105014.166}
SPL {X  -137.187, Y  +758.820, Z    +0.000, E1   -72.156, E3 +105020.169}
SPL {X  -134.014, Y  +763.891, Z    +0.000, E1   -71.759, E3 +105025.855}
SPL {X  -130.657, Y  +768.834, Z    +0.000, E1   -71.330, E3 +105031.470}
SPL {X  -126.020, Y  +775.068, Z    +0.000, E1   -70.718, E3 +105038.598}
SPL {X  -121.287, Y  +780.838, Z    +0.000, E1   -70.013, E3 +105045.172}
SPL {X   -75.772, Y  +817.409, Z    +0.000, E1   -56.226, E3 +105172.524}
ENDSPLINE

SPLINE
SPL {X  -124.054, Y  +777.532, Z    +0.000, E1   -54.436, E3 +105355.752}
SPL {X  -145.922, Y  +742.101, Z    +0.000, E1   -46.535, E3 +105374.021}
SPL {X  -155.216, Y  +715.293, Z    +0.000, E1   -34.460, E3 +105380.214}
SPL {X  -158.715, Y  +696.660, Z    +0.000, E1   -21.368, E3 +105382.541}
SPL {X  -159.838, Y  +683.473, Z    +0.000, E1    -9.532, E3 +105383.337}
SPL {X  -159.990, Y  +674.579, Z    +0.000, E1    -0.168, E3 +105383.520}
SPL {X  -159.990, Y  +672.677, Z    +0.000, E1    +3.879, E3 +105383.536}
SPL {X  -159.990, Y  +669.117, Z    +0.000, E1   +12.900, E3 +105383.618}
SPL {X  -159.990, Y  +663.639, Z    +0.000, E1   +26.675, E3 +105383.904}
SPL {X  -159.990, Y  +656.057, Z    +0.000, E1   +43.288, E3 +105384.560}
SPL {X  -159.990, Y  +647.797, Z    +0.000, E1   +54.469, E3 +105385.697}
SPL {X  -159.990, Y  +630.178, Z    +0.000, E1   +65.480, E3 +105389.381}
SPL {X  -159.990, Y  +547.268, Z    +0.000, E1   +73.735, E3 +105416.665}
SPL {X  -159.091, Y  +360.560, Z    +0.000, E1   +74.726, E3 +105502.991}
SPL {X  -156.418, Y  +343.879, Z    +0.000, E1   +74.473, E3 +105515.417}
SPL {X  -153.414, Y  +332.103, Z    +0.000, E1   +74.378, E3 +105523.091}
SPL {X  -141.909, Y  +303.617, Z    +0.000, E1   +76.515, E3 +105515.621}
ENDSPLINE

SPLINE
SPL {X  -142.567, Y  +304.895, Z    +0.000, E1   +75.566, E3 +105524.437}
ENDSPLINE

SPLINE
SPL {X  -141.999, Y  +303.790, Z    +0.000, E1   +74.633, E3 +105533.688}
SPL {X  -141.780, Y  +303.371, Z    +0.000, E1   +73.549, E3 +105543.262}
SPL {X  -140.619, Y  +301.190, Z    +0.000, E1   +72.741, E3 +105551.108}
SPL {X  -137.438, Y  +295.601, Z    +0.000, E1   +72.365, E3 +105557.196}
SPL {X  -134.156, Y  +290.328, Z    +0.000, E1   +71.962, E3 +105563.068}
SPL {X  -130.677, Y  +285.194, Z    +0.000, E1   +71.519, E3 +105568.873}
SPL {X  -126.239, Y  +279.212, Z    +0.000, E1   +70.937, E3 +105575.674}
SPL {X  -121.335, Y  +273.218, Z    +0.000, E1   +70.225, E3 +105582.462}
SPL {X   -79.311, Y  +238.552, Z    +0.000, E1   +58.563, E3 +105678.939}
ENDSPLINE

SPLINE
SPL {X  -105.077, Y  +256.854, Z    +0.000, E1   +55.187, E3 +105866.491}
SPL {X  -133.208, Y  +288.886, Z    +0.000, E1   +52.003, E3 +105899.592}
SPL {X  -149.825, Y  +321.381, Z    +0.000, E1   +42.580, E3 +105912.746}
SPL {X  -156.491, Y  +344.222, Z    +0.000, E1   +30.612, E3 +105917.252}
SPL {X  -159.275, Y  +362.387, Z    +0.000, E1   +16.907, E3 +105919.166}
SPL {X  -159.964, Y  +374.630, Z    +0.000, E1    +5.249, E3 +105919.739}
SPL {X  -159.990, Y  +379.484, Z    +0.000, E1    +0.034, E3 +105919.795}
SPL {X  -159.990, Y  +381.639, Z    +0.000, E1    -4.454, E3 +105919.817}
SPL {X  -159.990, Y  +385.871, Z    +0.000, E1   -15.161, E3 +105919.933}
SPL {X  -159.990, Y  +391.065, Z    +0.000, E1   -28.187, E3 +105920.221}
SPL {X  -159.990, Y  +397.286, Z    +0.000, E1   -41.591, E3 +105920.764}
SPL {X  -159.990, Y  +406.369, Z    +0.000, E1   -54.148, E3 +105921.982}
SPL {X  -159.990, Y  +426.617, Z    +0.000, E1   -66.230, E3 +105926.232}
SPL {X  -159.990, Y  +499.521, Z    +0.000, E1   -73.662, E3 +105949.559}
SPL {X  -159.629, Y  +687.249, Z    +0.000, E1   -74.539, E3 +106037.443}
SPL {X  -157.983, Y  +701.765, Z    +0.000, E1   -74.384, E3 +106047.675}
SPL {X  -155.520, Y  +714.054, Z    +0.000, E1   -74.151, E3 +106057.429}
SPL {X  -152.569, Y  +724.660, Z    +0.000, E1   -73.857, E3 +106066.664}
SPL {X  -149.625, Y  +733.149, Z    +0.000, E1   -73.553, E3 +106074.599}
SPL {X  -146.617, Y  +740.532, Z    +0.000, E1   -73.233, E3 +106081.875}
SPL {X  -143.394, Y  +747.457, Z    +0.000, E1   -72.883, E3 +106088.972}
SPL {X  -140.332, Y  +753.336, Z    +0.000, E1   -72.527, E3 +106095.247}
SPL {X  -137.187, Y  +758.820, Z    +0.000, E1   -72.156, E3 +106101.250}
SPL {X  -134.014, Y  +763.891, Z    +0.000, E1   -71.759, E3 +106106.936}
SPL {X  -130.657, Y  +768.834, Z    +0.000, E1   -71.330, E3 +106112.551}
SPL {X  -126.020, Y  +775.068, Z    +0.000, E1   -70.718, E3 +106119.679}
SPL {X  -121.287, Y  +780.838, Z    +0.000, E1   -70.013, E3 +106126.253}
SPL {X   -75.772, Y  +817.409, Z    +0.000, E1   -56.226, E3 +106253.605}
ENDSPLINE

